LIN {X 0,Y 185.683,Z 170.354,A -85,B 0,C 180,E1 -22212.634,E2 -22212.634} C_VEL
LIN {X 0,Y 186.754,Z 173.291,A -85,B 0,C 180,E1 -22212.96,E2 -22212.96} C_VEL
LIN {X 0,Y 193.586,Z 186.24,A -85,B 0,C 180,E1 -22214.699,E2 -22214.699} C_VEL
LIN {X 0,Y 199.796,Z 199.622,A -85,B 0,C 180,E1 -22216.226,E2 -22216.226} C_VEL
LIN {X 0,Y 202.678,Z 207.739,A -85,B 0,C 180,E1 -22216.973,E2 -22216.973} C_VEL
LIN {X 0,Y 199.951,Z 270.572,A -85,B 0,C 180,E1 -22219.192,E2 -22219.192} C_VEL
LIN {X 0,Y 198.885,Z 284.057,A -85,B 0,C 180,E1 -22220.081,E2 -22220.081} C_VEL
LIN {X 0,Y 197.521,Z 296.496,A -85,B 0,C 180,E1 -22221.303,E2 -22221.303} C_VEL
LIN {X 0,Y 195.797,Z 307.712,A -85,B 0,C 180,E1 -22222.783,E2 -22222.783} C_VEL
LIN {X 0,Y 193.672,Z 319.403,A -85,B 0,C 180,E1 -22224.795,E2 -22224.795} C_VEL
LIN {X 0,Y 191.562,Z 329.915,A -85,B 0,C 180,E1 -22227.109,E2 -22227.109} C_VEL
LIN {X 0,Y 189.509,Z 339.066,A -85,B 0,C 180,E1 -22229.646,E2 -22229.646} C_VEL
LIN {X 0,Y 187.491,Z 347.803,A -85,B 0,C 180,E1 -22232.686,E2 -22232.686} C_VEL
LIN {X 0,Y 185.853,Z 355.279,A -85,B 0,C 180,E1 -22235.969,E2 -22235.969} C_VEL
LIN {X 0,Y 184.768,Z 360.328,A -85,B 0,C 180,E1 -22238.752,E2 -22238.752} C_VEL
LIN {X 0,Y 183.841,Z 365.228,A -85,B 0,C 180,E1 -22242.138,E2 -22242.138} C_VEL
LIN {X 0,Y 183.252,Z 368.971,A -85,B 0,C 180,E1 -22245.573,E2 -22245.573} C_VEL
LIN {X 0,Y 183.005,Z 370.856,A -85,B 0,C 180,E1 -22247.893,E2 -22247.893} C_VEL
LIN {X 0,Y 182.982,Z 372.28,A -85,B 0,C 180,E1 -22250.223,E2 -22250.223} C_VEL
LIN {X 0,Y 183.211,Z 373.408,A -85,B 0,C 180,E1 -22252.981,E2 -22252.981} C_VEL
LIN {X 0,Y 184.045,Z 373.895,A -85,B 0,C 180,E1 -22257.274,E2 -22257.274} C_VEL
LIN {X 0,Y 184.848,Z 373.552,A -85,B 0,C 180,E1 -22259.622,E2 -22259.622} C_VEL
LIN {X 0,Y 185.845,Z 372.724,A -85,B 0,C 180,E1 -22261.967,E2 -22261.967} C_VEL
LIN {X 0,Y 187.135,Z 371.423,A -85,B 0,C 180,E1 -22264.287,E2 -22264.287} C_VEL
LIN {X 0,Y 189.469,Z 368.561,A -85,B 0,C 180,E1 -22267.737,E2 -22267.737} C_VEL
LIN {X 0,Y 192.379,Z 364.501,A -85,B 0,C 180,E1 -22271.116,E2 -22271.116} C_VEL
LIN {X 0,Y 196.276,Z 358.58,A -85,B 0,C 180,E1 -22274.64,E2 -22274.64} C_VEL
LIN {X 0,Y 200.108,Z 352.117,A -85,B 0,C 180,E1 -22277.523,E2 -22277.523} C_VEL
LIN {X 0,Y 204.75,Z 343.271,A -85,B 0,C 180,E1 -22280.562,E2 -22280.562} C_VEL
LIN {X 0,Y 209,Z 334.332,A -85,B 0,C 180,E1 -22282.876,E2 -22282.876} C_VEL
LIN {X 0,Y 213.308,Z 323.651,A -85,B 0,C 180,E1 -22285.043,E2 -22285.043} C_VEL
LIN {X 0,Y 216.807,Z 313.421,A -85,B 0,C 180,E1 -22286.659,E2 -22286.659} C_VEL
LIN {X 0,Y 219.931,Z 301.93,A -85,B 0,C 180,E1 -22288.084,E2 -22288.084} C_VEL
LIN {X 0,Y 222.4,Z 290.554,A -85,B 0,C 180,E1 -22289.133,E2 -22289.133} C_VEL
LIN {X 0,Y 224.406,Z 278.014,A -85,B 0,C 180,E1 -22289.955,E2 -22289.955} C_VEL
LIN {X 0,Y 225.625,Z 265.738,A -85,B 0,C 180,E1 -22290.474,E2 -22290.474} C_VEL
LIN {X 0,Y 227.824,Z 230.741,A -85,B 0,C 180,E1 -22291.554,E2 -22291.554} C_VEL
LIN {X 0,Y 224.167,Z 223.088,A -85,B 0,C 180,E1 -22293.044,E2 -22293.044} C_VEL
LIN {X 0,Y 217.84,Z 212.554,A -85,B 0,C 180,E1 -22295.719,E2 -22295.719} C_VEL
LIN {X 0,Y 212.058,Z 203.914,A -85,B 0,C 180,E1 -22298.467,E2 -22298.467} C_VEL
LIN {X 0,Y 206.963,Z 196.712,A -85,B 0,C 180,E1 -22301.18,E2 -22301.18} C_VEL
LIN {X 0,Y 204.092,Z 192.954,A -85,B 0,C 180,E1 -22302.853,E2 -22302.853} C_VEL
LIN {X 0,Y 200.713,Z 188.672,A -85,B 0,C 180,E1 -22305.051,E2 -22305.051} C_VEL
LIN {X 0,Y 199.927,Z 187.365,A -85,B 0,C 180,E1 -22305.625,E2 -22305.625} C_VEL
LIN {X 0,Y 197.269,Z 184.822,A -85,B 0,C 180,E1 -22307.527,E2 -22307.527} C_VEL
LIN {X 0,Y 195.63,Z 181.953,A -85,B 0,C 180,E1 -22308.932,E2 -22308.932} C_VEL
LIN {X 0,Y 192.955,Z 179.723,A -85,B 0,C 180,E1 -22311.217,E2 -22311.217} C_VEL
LIN {X 0,Y 191.565,Z 177.134,A -85,B 0,C 180,E1 -22312.756,E2 -22312.756} C_VEL
LIN {X 0,Y 191.264,Z 176.32,A -85,B 0,C 180,E1 -22313.143,E2 -22313.143} C_VEL
LIN {X 0,Y 188.409,Z 174.865,A -85,B 0,C 180,E1 -22316.391,E2 -22316.391} C_VEL
LIN {X 0,Y 186.674,Z 171.895,A -85,B 0,C 180,E1 -22319.259,E2 -22319.259} C_VEL
LIN {X 0,Y 186.346,Z 170.267,A -85,B 0,C 180,E1 -22320.135,E2 -22320.135} C_VEL
LIN {X 0,Y 185.885,Z 170.317,A -85,B 0,C 180,E1 -22324.337,E2 -22324.337} C_VEL
LIN {X 0,Y 185.976,Z 170.302,A -85,B 0,C 180,E1 -22328.695,E2 -22328.695} C_VEL
LIN {X 0,Y 185.723,Z 170.332,A -85,B 0,C 180,E1 -22333.124,E2 -22333.124} C_VEL
LIN {X 0,Y 185.682,Z 170.347,A -85,B 0,C 180,E1 -22336.492,E2 -22336.492} C_VEL
LIN {X 0,Y 185.915,Z 171.497,A -85,B 0,C 180,E1 -22338.814,E2 -22338.814} C_VEL
LIN {X 0,Y 186.795,Z 173.557,A -85,B 0,C 180,E1 -22340.655,E2 -22340.655} C_VEL
LIN {X 0,Y 188.885,Z 175.776,A -85,B 0,C 180,E1 -22343.723,E2 -22343.723} C_VEL
LIN {X 0,Y 191.922,Z 179.165,A -85,B 0,C 180,E1 -22347.242,E2 -22347.242} C_VEL
LIN {X 0,Y 194.898,Z 183.776,A -85,B 0,C 180,E1 -22350.131,E2 -22350.131} C_VEL
LIN {X 0,Y 197.691,Z 187.166,A -85,B 0,C 180,E1 -22352.379,E2 -22352.379} C_VEL
LIN {X 0,Y 202.172,Z 193.838,A -85,B 0,C 180,E1 -22355.611,E2 -22355.611} C_VEL
LIN {X 0,Y 206.17,Z 199.973,A -85,B 0,C 180,E1 -22358.086,E2 -22358.086} C_VEL
LIN {X 0,Y 209.889,Z 206.05,A -85,B 0,C 180,E1 -22360.173,E2 -22360.173} C_VEL
LIN {X 0,Y 213.804,Z 212.78,A -85,B 0,C 180,E1 -22362.196,E2 -22362.196} C_VEL
LIN {X 0,Y 219.154,Z 223.042,A -85,B 0,C 180,E1 -22364.732,E2 -22364.732} C_VEL
LIN {X 0,Y 224.276,Z 234.48,A -85,B 0,C 180,E1 -22366.986,E2 -22366.986} C_VEL
LIN {X 0,Y 226.38,Z 239.916,A -85,B 0,C 180,E1 -22367.89,E2 -22367.89} C_VEL
LIN {X 0,Y 226.931,Z 246.644,A -85,B 0,C 180,E1 -22368.381,E2 -22368.381} C_VEL
LIN {X 0,Y 225.009,Z 277.037,A -85,B 0,C 180,E1 -22369.312,E2 -22369.312} C_VEL
LIN {X 0,Y 224.097,Z 282.869,A -85,B 0,C 180,E1 -22369.364,E2 -22369.364} C_VEL
LIN {X 0,Y 221.088,Z 292.299,A -85,B 0,C 180,E1 -22369.24,E2 -22369.24} C_VEL
LIN {X 0,Y 217.548,Z 301.55,A -85,B 0,C 180,E1 -22369.224,E2 -22369.224} C_VEL
LIN {X 0,Y 215.797,Z 307.1,A -85,B 0,C 180,E1 -22369.487,E2 -22369.487} C_VEL
LIN {X 0,Y 212.279,Z 320.078,A -85,B 0,C 180,E1 -22370.715,E2 -22370.715} C_VEL
LIN {X 0,Y 208.678,Z 330.767,A -85,B 0,C 180,E1 -22372.074,E2 -22372.074} C_VEL
LIN {X 0,Y 204.289,Z 341.732,A -85,B 0,C 180,E1 -22373.904,E2 -22373.904} C_VEL
LIN {X 0,Y 199.37,Z 352.427,A -85,B 0,C 180,E1 -22376.275,E2 -22376.275} C_VEL
LIN {X 0,Y 195.224,Z 360.362,A -85,B 0,C 180,E1 -22378.533,E2 -22378.533} C_VEL
LIN {X 0,Y 190.711,Z 368.187,A -85,B 0,C 180,E1 -22381.375,E2 -22381.375} C_VEL
LIN {X 0,Y 186.739,Z 374.659,A -85,B 0,C 180,E1 -22384.473,E2 -22384.473} C_VEL
LIN {X 0,Y 183.642,Z 379.535,A -85,B 0,C 180,E1 -22387.498,E2 -22387.498} C_VEL
LIN {X 0,Y 180.899,Z 383.498,A -85,B 0,C 180,E1 -22390.717,E2 -22390.717} C_VEL
LIN {X 0,Y 178.676,Z 386.462,A -85,B 0,C 180,E1 -22394.017,E2 -22394.017} C_VEL
LIN {X 0,Y 176.939,Z 388.948,A -85,B 0,C 180,E1 -22398.545,E2 -22398.545} C_VEL
LIN {X 0,Y 176.128,Z 389.914,A -85,B 0,C 180,E1 -22403.124,E2 -22403.124} C_VEL
LIN {X 0,Y 176.125,Z 389.685,A -85,B 0,C 180,E1 -22406.027,E2 -22406.027} C_VEL
LIN {X 0,Y 176.394,Z 388.365,A -85,B 0,C 180,E1 -22410,E2 -22410} C_VEL
LIN {X 0,Y 176.229,Z 387.022,A -85,B 0,C 180,E1 -22412.285,E2 -22412.285} C_VEL
LIN {X 0,Y 176.169,Z 384.135,A -85,B 0,C 180,E1 -22415.723,E2 -22415.723} C_VEL
LIN {X 0,Y 176.448,Z 380.179,A -85,B 0,C 180,E1 -22419.167,E2 -22419.167} C_VEL
LIN {X 0,Y 177.299,Z 374.04,A -85,B 0,C 180,E1 -22423.175,E2 -22423.175} C_VEL
LIN {X 0,Y 178.698,Z 367.3,A -85,B 0,C 180,E1 -22426.566,E2 -22426.566} C_VEL
LIN {X 0,Y 180.547,Z 358.895,A -85,B 0,C 180,E1 -22429.913,E2 -22429.913} C_VEL
LIN {X 0,Y 181.898,Z 352.509,A -85,B 0,C 180,E1 -22431.983,E2 -22431.983} C_VEL
LIN {X 0,Y 183.957,Z 344.092,A -85,B 0,C 180,E1 -22434.248,E2 -22434.248} C_VEL
LIN {X 0,Y 186.267,Z 333.179,A -85,B 0,C 180,E1 -22436.618,E2 -22436.618} C_VEL
LIN {X 0,Y 188.393,Z 322.564,A -85,B 0,C 180,E1 -22438.401,E2 -22438.401} C_VEL
LIN {X 0,Y 190.53,Z 309.778,A -85,B 0,C 180,E1 -22440.018,E2 -22440.018} C_VEL
LIN {X 0,Y 192.193,Z 297.008,A -85,B 0,C 180,E1 -22441.175,E2 -22441.175} C_VEL
LIN {X 0,Y 193.255,Z 284.752,A -85,B 0,C 180,E1 -22441.9,E2 -22441.9} C_VEL
LIN {X 0,Y 195.225,Z 238.101,A -85,B 0,C 180,E1 -22443.6,E2 -22443.6} C_VEL
LIN {X 0,Y 192.063,Z 207.786,A -85,B 0,C 180,E1 -22445.365,E2 -22445.365} C_VEL
LIN {X 0,Y 185.656,Z 190.417,A -85,B 0,C 180,E1 -22447.212,E2 -22447.212} C_VEL
LIN {X 0,Y 180.83,Z 179.385,A -85,B 0,C 180,E1 -22448.597,E2 -22448.597} C_VEL
LIN {X 0,Y 179.797,Z 176.7,A -85,B 0,C 180,E1 -22449.002,E2 -22449.002} C_VEL
LIN {X 0,Y 178.427,Z 171.261,A -85,B 0,C 180,E1 -22452.036,E2 -22452.036} C_VEL
LIN {X 0,Y 178.395,Z 171.266,A -85,B 0,C 180,E1 -22455.163,E2 -22455.163} C_VEL
LIN {X 0,Y 178.404,Z 171.265,A -85,B 0,C 180,E1 -22458.458,E2 -22458.458} C_VEL
LIN {X 0,Y 178.423,Z 171.263,A -85,B 0,C 180,E1 -22463.783,E2 -22463.783} C_VEL
LIN {X 0,Y 178.488,Z 171.252,A -85,B 0,C 180,E1 -22466.546,E2 -22466.546} C_VEL
LIN {X 0,Y 178.524,Z 171.248,A -85,B 0,C 180,E1 -22470.006,E2 -22470.006} C_VEL
LIN {X 0,Y 178.52,Z 171.248,A -85,B 0,C 180,E1 -22474.885,E2 -22474.885} C_VEL
LIN {X 0,Y 178.589,Z 171.197,A -85,B 0,C 180,E1 -22480.815,E2 -22480.815} C_VEL
LIN {X 0,Y 178.643,Z 171.22,A -85,B 0,C 180,E1 -22486.346,E2 -22486.346} C_VEL
LIN {X 0,Y 178.905,Z 171.195,A -85,B 0,C 180,E1 -22490.959,E2 -22490.959} C_VEL
LIN {X 0,Y 179.149,Z 171.165,A -85,B 0,C 180,E1 -22497.751,E2 -22497.751} C_VEL
LIN {X 0,Y 179.37,Z 171.135,A -85,B 0,C 180,E1 -22500,E2 -22500} C_VEL
LIN {X 0,Y 178.867,Z 171.194,A -85,B 0,C 180,E1 -22504.507,E2 -22504.507} C_VEL
LIN {X 0,Y 178.911,Z 171.191,A -85,B 0,C 180,E1 -22509.04,E2 -22509.04} C_VEL
LIN {X 0,Y 178.657,Z 171.222,A -85,B 0,C 180,E1 -22513.652,E2 -22513.652} C_VEL
LIN {X 0,Y 178.622,Z 171.227,A -85,B 0,C 180,E1 -22519.215,E2 -22519.215} C_VEL
LIN {X 0,Y 178.519,Z 171.246,A -85,B 0,C 180,E1 -22525.114,E2 -22525.114} C_VEL
LIN {X 0,Y 178.52,Z 171.232,A -85,B 0,C 180,E1 -22529.993,E2 -22529.993} C_VEL
LIN {X 0,Y 178.483,Z 171.25,A -85,B 0,C 180,E1 -22534.219,E2 -22534.219} C_VEL
LIN {X 0,Y 178.394,Z 171.25,A -85,B 0,C 180,E1 -22539.074,E2 -22539.074} C_VEL
LIN {X 0,Y 178.397,Z 171.261,A -85,B 0,C 180,E1 -22542.045,E2 -22542.045} C_VEL
LIN {X 0,Y 178.393,Z 171.253,A -85,B 0,C 180,E1 -22545.164,E2 -22545.164} C_VEL
LIN {X 0,Y 178.402,Z 171.261,A -85,B 0,C 180,E1 -22548.459,E2 -22548.459} C_VEL
LIN {X 0,Y 178.422,Z 171.261,A -85,B 0,C 180,E1 -22553.783,E2 -22553.783} C_VEL
LIN {X 0,Y 178.486,Z 171.242,A -85,B 0,C 180,E1 -22556.547,E2 -22556.547} C_VEL
LIN {X 0,Y 178.522,Z 171.233,A -85,B 0,C 180,E1 -22560.006,E2 -22560.006} C_VEL
LIN {X 0,Y 178.519,Z 171.237,A -85,B 0,C 180,E1 -22564.886,E2 -22564.886} C_VEL
LIN {X 0,Y 178.624,Z 171.226,A -85,B 0,C 180,E1 -22571.288,E2 -22571.288} C_VEL
LIN {X 0,Y 179.695,Z 174.19,A -85,B 0,C 180,E1 -22571.687,E2 -22571.687} C_VEL
LIN {X 0,Y 184.03,Z 181.923,A -85,B 0,C 180,E1 -22572.86,E2 -22572.86} C_VEL
LIN {X 0,Y 192.925,Z 200.17,A -85,B 0,C 180,E1 -22575.192,E2 -22575.192} C_VEL
LIN {X 0,Y 196.304,Z 209.181,A -85,B 0,C 180,E1 -22576.1,E2 -22576.1} C_VEL
LIN {X 0,Y 193.535,Z 270.405,A -85,B 0,C 180,E1 -22578.313,E2 -22578.313} C_VEL
LIN {X 0,Y 192.39,Z 284.408,A -85,B 0,C 180,E1 -22579.257,E2 -22579.257} C_VEL
LIN {X 0,Y 190.855,Z 297.508,A -85,B 0,C 180,E1 -22580.596,E2 -22580.596} C_VEL
LIN {X 0,Y 188.946,Z 309.37,A -85,B 0,C 180,E1 -22582.251,E2 -22582.251} C_VEL
LIN {X 0,Y 186.759,Z 320.819,A -85,B 0,C 180,E1 -22584.331,E2 -22584.331} C_VEL
LIN {X 0,Y 184.559,Z 331.091,A -85,B 0,C 180,E1 -22586.726,E2 -22586.726} C_VEL
LIN {X 0,Y 182.317,Z 340.478,A -85,B 0,C 180,E1 -22589.481,E2 -22589.481} C_VEL
LIN {X 0,Y 180.259,Z 349.401,A -85,B 0,C 180,E1 -22592.794,E2 -22592.794} C_VEL
LIN {X 0,Y 178.58,Z 356.596,A -85,B 0,C 180,E1 -22596.213,E2 -22596.213} C_VEL
LIN {X 0,Y 177.519,Z 361.503,A -85,B 0,C 180,E1 -22599.112,E2 -22599.112} C_VEL
LIN {X 0,Y 176.617,Z 366.201,A -85,B 0,C 180,E1 -22602.642,E2 -22602.642} C_VEL
LIN {X 0,Y 176.025,Z 370.083,A -85,B 0,C 180,E1 -22606.62,E2 -22606.62} C_VEL
LIN {X 0,Y 175.943,Z 372.894,A -85,B 0,C 180,E1 -22611.07,E2 -22611.07} C_VEL
LIN {X 0,Y 176.181,Z 373.768,A -85,B 0,C 180,E1 -22613.51,E2 -22613.51} C_VEL
LIN {X 0,Y 176.593,Z 374.196,A -85,B 0,C 180,E1 -22615.963,E2 -22615.963} C_VEL
LIN {X 0,Y 177.676,Z 374.027,A -85,B 0,C 180,E1 -22619.518,E2 -22619.518} C_VEL
LIN {X 0,Y 179.353,Z 372.789,A -85,B 0,C 180,E1 -22623.271,E2 -22623.271} C_VEL
LIN {X 0,Y 180.795,Z 371.406,A -85,B 0,C 180,E1 -22625.669,E2 -22625.669} C_VEL
LIN {X 0,Y 183.351,Z 368.412,A -85,B 0,C 180,E1 -22629.18,E2 -22629.18} C_VEL
LIN {X 0,Y 186.612,Z 364.099,A -85,B 0,C 180,E1 -22632.68,E2 -22632.68} C_VEL
LIN {X 0,Y 190.53,Z 358.405,A -85,B 0,C 180,E1 -22636.038,E2 -22636.038} C_VEL
LIN {X 0,Y 194.945,Z 351.263,A -85,B 0,C 180,E1 -22639.208,E2 -22639.208} C_VEL
LIN {X 0,Y 199.065,Z 343.785,A -85,B 0,C 180,E1 -22641.771,E2 -22641.771} C_VEL
LIN {X 0,Y 203.726,Z 334.428,A -85,B 0,C 180,E1 -22644.224,E2 -22644.224} C_VEL
LIN {X 0,Y 207.99,Z 324.269,A -85,B 0,C 180,E1 -22646.314,E2 -22646.314} C_VEL
LIN {X 0,Y 211.87,Z 313.396,A -85,B 0,C 180,E1 -22648.047,E2 -22648.047} C_VEL
LIN {X 0,Y 215.169,Z 301.7,A -85,B 0,C 180,E1 -22649.484,E2 -22649.484} C_VEL
LIN {X 0,Y 217.846,Z 289.592,A -85,B 0,C 180,E1 -22650.582,E2 -22650.582} C_VEL
LIN {X 0,Y 219.859,Z 276.83,A -85,B 0,C 180,E1 -22651.4,E2 -22651.4} C_VEL
LIN {X 0,Y 221.194,Z 262.498,A -85,B 0,C 180,E1 -22651.941,E2 -22651.941} C_VEL
LIN {X 0,Y 223.096,Z 233.455,A -85,B 0,C 180,E1 -22652.844,E2 -22652.844} C_VEL
LIN {X 0,Y 219.833,Z 226.818,A -85,B 0,C 180,E1 -22654.245,E2 -22654.245} C_VEL
LIN {X 0,Y 214.285,Z 217.443,A -85,B 0,C 180,E1 -22656.756,E2 -22656.756} C_VEL
LIN {X 0,Y 208.779,Z 209.045,A -85,B 0,C 180,E1 -22659.527,E2 -22659.527} C_VEL
LIN {X 0,Y 204.268,Z 202.61,A -85,B 0,C 180,E1 -22662.058,E2 -22662.058} C_VEL
LIN {X 0,Y 200.956,Z 198.121,A -85,B 0,C 180,E1 -22664.144,E2 -22664.144} C_VEL
LIN {X 0,Y 198.215,Z 194.314,A -85,B 0,C 180,E1 -22666.072,E2 -22666.072} C_VEL
LIN {X 0,Y 194.988,Z 190.63,A -85,B 0,C 180,E1 -22668.538,E2 -22668.538} C_VEL
LIN {X 0,Y 193.865,Z 188.579,A -85,B 0,C 180,E1 -22669.557,E2 -22669.557} C_VEL
LIN {X 0,Y 191.372,Z 186.351,A -85,B 0,C 180,E1 -22671.811,E2 -22671.811} C_VEL
LIN {X 0,Y 189.821,Z 183.428,A -85,B 0,C 180,E1 -22673.623,E2 -22673.623} C_VEL
LIN {X 0,Y 186.829,Z 181.328,A -85,B 0,C 180,E1 -22677.305,E2 -22677.305} C_VEL
LIN {X 0,Y 185.305,Z 178.253,A -85,B 0,C 180,E1 -22680.136,E2 -22680.136} C_VEL
LIN {X 0,Y 185.063,Z 177.272,A -85,B 0,C 180,E1 -22680.816,E2 -22680.816} C_VEL
LIN {X 0,Y 182.802,Z 176.663,A -85,B 0,C 180,E1 -22688.847,E2 -22688.847} C_VEL
LIN {X 0,Y 184.131,Z 177.385,A -85,B 0,C 180,E1 -22696.635,E2 -22696.635} C_VEL
LIN {X 0,Y 184.769,Z 178.417,A -85,B 0,C 180,E1 -22698.331,E2 -22698.331} C_VEL
LIN {X 0,Y 185.917,Z 180.829,A -85,B 0,C 180,E1 -22700.757,E2 -22700.757} C_VEL
LIN {X 0,Y 187.603,Z 182.649,A -85,B 0,C 180,E1 -22703.284,E2 -22703.284} C_VEL
LIN {X 0,Y 190.562,Z 186.17,A -85,B 0,C 180,E1 -22706.859,E2 -22706.859} C_VEL
LIN {X 0,Y 193.141,Z 190.298,A -85,B 0,C 180,E1 -22709.484,E2 -22709.484} C_VEL
LIN {X 0,Y 195.738,Z 193.586,A -85,B 0,C 180,E1 -22711.677,E2 -22711.677} C_VEL
LIN {X 0,Y 199.913,Z 200.03,A -85,B 0,C 180,E1 -22714.84,E2 -22714.84} C_VEL
LIN {X 0,Y 203.71,Z 206.099,A -85,B 0,C 180,E1 -22717.331,E2 -22717.331} C_VEL
LIN {X 0,Y 206.999,Z 211.66,A -85,B 0,C 180,E1 -22719.273,E2 -22719.273} C_VEL
LIN {X 0,Y 211.426,Z 219.589,A -85,B 0,C 180,E1 -22721.669,E2 -22721.669} C_VEL
LIN {X 0,Y 216.84,Z 230.662,A -85,B 0,C 180,E1 -22724.358,E2 -22724.358} C_VEL
LIN {X 0,Y 221.216,Z 241.243,A -85,B 0,C 180,E1 -22726.381,E2 -22726.381} C_VEL
LIN {X 0,Y 221.895,Z 242.935,A -85,B 0,C 180,E1 -22726.683,E2 -22726.683} C_VEL
LIN {X 0,Y 222.294,Z 247.076,A -85,B 0,C 180,E1 -22727.02,E2 -22727.02} C_VEL
LIN {X 0,Y 219.532,Z 285.815,A -85,B 0,C 180,E1 -22728.25,E2 -22728.25} C_VEL
LIN {X 0,Y 217.473,Z 299.233,A -85,B 0,C 180,E1 -22728.932,E2 -22728.932} C_VEL
LIN {X 0,Y 215.797,Z 307.1,A -85,B 0,C 180,E1 -22729.487,E2 -22729.487} C_VEL
LIN {X 0,Y 213.849,Z 312.694,A -85,B 0,C 180,E1 -22729.811,E2 -22729.811} C_VEL
LIN {X 0,Y 209.199,Z 321.494,A -85,B 0,C 180,E1 -22730.134,E2 -22730.134} C_VEL
LIN {X 0,Y 204.327,Z 329.786,A -85,B 0,C 180,E1 -22730.653,E2 -22730.653} C_VEL
LIN {X 0,Y 202.043,Z 334.607,A -85,B 0,C 180,E1 -22731.281,E2 -22731.281} C_VEL
LIN {X 0,Y 197.677,Z 344.642,A -85,B 0,C 180,E1 -22733.133,E2 -22733.133} C_VEL
LIN {X 0,Y 192.711,Z 354.666,A -85,B 0,C 180,E1 -22735.578,E2 -22735.578} C_VEL
LIN {X 0,Y 187.604,Z 363.522,A -85,B 0,C 180,E1 -22738.367,E2 -22738.367} C_VEL
LIN {X 0,Y 183.06,Z 370.68,A -85,B 0,C 180,E1 -22741.321,E2 -22741.321} C_VEL
LIN {X 0,Y 179.28,Z 376.429,A -85,B 0,C 180,E1 -22744.455,E2 -22744.455} C_VEL
LIN {X 0,Y 176.033,Z 381.002,A -85,B 0,C 180,E1 -22747.71,E2 -22747.71} C_VEL
LIN {X 0,Y 173.346,Z 384.521,A -85,B 0,C 180,E1 -22751.074,E2 -22751.074} C_VEL
LIN {X 0,Y 171.842,Z 386.314,A -85,B 0,C 180,E1 -22753.364,E2 -22753.364} C_VEL
LIN {X 0,Y 169.967,Z 388.718,A -85,B 0,C 180,E1 -22758.068,E2 -22758.068} C_VEL
LIN {X 0,Y 169.371,Z 389.351,A -85,B 0,C 180,E1 -22760.445,E2 -22760.445} C_VEL
LIN {X 0,Y 169.079,Z 389.581,A -85,B 0,C 180,E1 -22762.836,E2 -22762.836} C_VEL
LIN {X 0,Y 169.144,Z 388.853,A -85,B 0,C 180,E1 -22767.618,E2 -22767.618} C_VEL
LIN {X 0,Y 169.309,Z 387.903,A -85,B 0,C 180,E1 -22770,E2 -22770} C_VEL
LIN {X 0,Y 169.1,Z 385.236,A -85,B 0,C 180,E1 -22774.07,E2 -22774.07} C_VEL
LIN {X 0,Y 169.266,Z 380.947,A -85,B 0,C 180,E1 -22778.355,E2 -22778.355} C_VEL
LIN {X 0,Y 169.863,Z 376.113,A -85,B 0,C 180,E1 -22781.939,E2 -22781.939} C_VEL
LIN {X 0,Y 171.019,Z 369.981,A -85,B 0,C 180,E1 -22785.492,E2 -22785.492} C_VEL
LIN {X 0,Y 172.699,Z 362.32,A -85,B 0,C 180,E1 -22788.999,E2 -22788.999} C_VEL
LIN {X 0,Y 174.757,Z 353.387,A -85,B 0,C 180,E1 -22792.212,E2 -22792.212} C_VEL
LIN {X 0,Y 177.197,Z 343.797,A -85,B 0,C 180,E1 -22794.923,E2 -22794.923} C_VEL
LIN {X 0,Y 179.589,Z 332.885,A -85,B 0,C 180,E1 -22797.375,E2 -22797.375} C_VEL
LIN {X 0,Y 181.81,Z 322.285,A -85,B 0,C 180,E1 -22799.211,E2 -22799.211} C_VEL
LIN {X 0,Y 184.024,Z 309.51,A -85,B 0,C 180,E1 -22800.876,E2 -22800.876} C_VEL
LIN {X 0,Y 185.736,Z 296.808,A -85,B 0,C 180,E1 -22802.062,E2 -22802.062} C_VEL
LIN {X 0,Y 186.848,Z 284.399,A -85,B 0,C 180,E1 -22802.819,E2 -22802.819} C_VEL
LIN {X 0,Y 188.863,Z 238.895,A -85,B 0,C 180,E1 -22804.524,E2 -22804.524} C_VEL
LIN {X 0,Y 186.023,Z 210.18,A -85,B 0,C 180,E1 -22806.256,E2 -22806.256} C_VEL
LIN {X 0,Y 180.087,Z 193.89,A -85,B 0,C 180,E1 -22808.058,E2 -22808.058} C_VEL
LIN {X 0,Y 174.201,Z 180.352,A -85,B 0,C 180,E1 -22809.86,E2 -22809.86} C_VEL
LIN {X 0,Y 172.459,Z 176.4,A -85,B 0,C 180,E1 -22810.468,E2 -22810.468} C_VEL
LIN {X 0,Y 171.332,Z 172.144,A -85,B 0,C 180,E1 -22813.009,E2 -22813.009} C_VEL
LIN {X 0,Y 171.337,Z 172.146,A -85,B 0,C 180,E1 -22817.589,E2 -22817.589} C_VEL
LIN {X 0,Y 171.388,Z 172.139,A -85,B 0,C 180,E1 -22822.04,E2 -22822.04} C_VEL
LIN {X 0,Y 171.399,Z 172.136,A -85,B 0,C 180,E1 -22825.092,E2 -22825.092} C_VEL
LIN {X 0,Y 171.45,Z 172.129,A -85,B 0,C 180,E1 -22830.534,E2 -22830.534} C_VEL
LIN {X 0,Y 171.444,Z 172.128,A -85,B 0,C 180,E1 -22835.799,E2 -22835.799} C_VEL
LIN {X 0,Y 171.545,Z 172.072,A -85,B 0,C 180,E1 -22840.867,E2 -22840.867} C_VEL
LIN {X 0,Y 171.558,Z 172.097,A -85,B 0,C 180,E1 -22845.771,E2 -22845.771} C_VEL
LIN {X 0,Y 171.843,Z 172.077,A -85,B 0,C 180,E1 -22850.584,E2 -22850.584} C_VEL
LIN {X 0,Y 171.807,Z 172.073,A -85,B 0,C 180,E1 -22855.307,E2 -22855.307} C_VEL
LIN {X 0,Y 172.332,Z 172.011,A -85,B 0,C 180,E1 -22860,E2 -22860} C_VEL
LIN {X 0,Y 171.815,Z 172.074,A -85,B 0,C 180,E1 -22864.692,E2 -22864.692} C_VEL
LIN {X 0,Y 171.848,Z 172.07,A -85,B 0,C 180,E1 -22869.415,E2 -22869.415} C_VEL
LIN {X 0,Y 171.575,Z 172.106,A -85,B 0,C 180,E1 -22874.227,E2 -22874.227} C_VEL
LIN {X 0,Y 171.541,Z 172.106,A -85,B 0,C 180,E1 -22879.559,E2 -22879.559} C_VEL
LIN {X 0,Y 171.457,Z 172.126,A -85,B 0,C 180,E1 -22885.609,E2 -22885.609} C_VEL
LIN {X 0,Y 171.439,Z 172.113,A -85,B 0,C 180,E1 -22890.585,E2 -22890.585} C_VEL
LIN {X 0,Y 171.391,Z 172.132,A -85,B 0,C 180,E1 -22895.035,E2 -22895.035} C_VEL
LIN {X 0,Y 171.356,Z 172.125,A -85,B 0,C 180,E1 -22898.807,E2 -22898.807} C_VEL
LIN {X 0,Y 171.32,Z 172.135,A -85,B 0,C 180,E1 -22904.217,E2 -22904.217} C_VEL
LIN {X 0,Y 171.334,Z 172.142,A -85,B 0,C 180,E1 -22908.982,E2 -22908.982} C_VEL
LIN {X 0,Y 171.386,Z 172.13,A -85,B 0,C 180,E1 -22912.041,E2 -22912.041} C_VEL
LIN {X 0,Y 171.397,Z 172.134,A -85,B 0,C 180,E1 -22915.092,E2 -22915.092} C_VEL
LIN {X 0,Y 171.448,Z 172.119,A -85,B 0,C 180,E1 -22920.535,E2 -22920.535} C_VEL
LIN {X 0,Y 171.443,Z 172.115,A -85,B 0,C 180,E1 -22925.8,E2 -22925.8} C_VEL
LIN {X 0,Y 171.519,Z 172.118,A -85,B 0,C 180,E1 -22929.853,E2 -22929.853} C_VEL
LIN {X 0,Y 172.677,Z 175.19,A -85,B 0,C 180,E1 -22930.313,E2 -22930.313} C_VEL
LIN {X 0,Y 174.131,Z 177.575,A -85,B 0,C 180,E1 -22930.738,E2 -22930.738} C_VEL
LIN {X 0,Y 181.21,Z 190.789,A -85,B 0,C 180,E1 -22932.759,E2 -22932.759} C_VEL
LIN {X 0,Y 188.346,Z 206.211,A -85,B 0,C 180,E1 -22934.705,E2 -22934.705} C_VEL
LIN {X 0,Y 190.06,Z 211.072,A -85,B 0,C 180,E1 -22935.202,E2 -22935.202} C_VEL
LIN {X 0,Y 187.092,Z 271.113,A -85,B 0,C 180,E1 -22937.422,E2 -22937.422} C_VEL
LIN {X 0,Y 185.975,Z 284.449,A -85,B 0,C 180,E1 -22938.35,E2 -22938.35} C_VEL
LIN {X 0,Y 184.392,Z 297.494,A -85,B 0,C 180,E1 -22939.709,E2 -22939.709} C_VEL
LIN {X 0,Y 182.383,Z 309.432,A -85,B 0,C 180,E1 -22941.413,E2 -22941.413} C_VEL
LIN {X 0,Y 180.106,Z 320.927,A -85,B 0,C 180,E1 -22943.559,E2 -22943.559} C_VEL
LIN {X 0,Y 177.823,Z 331.246,A -85,B 0,C 180,E1 -22946.034,E2 -22946.034} C_VEL
LIN {X 0,Y 175.394,Z 341.035,A -85,B 0,C 180,E1 -22949.015,E2 -22949.015} C_VEL
LIN {X 0,Y 173.339,Z 349.607,A -85,B 0,C 180,E1 -22952.324,E2 -22952.324} C_VEL
LIN {X 0,Y 171.576,Z 356.834,A -85,B 0,C 180,E1 -22955.878,E2 -22955.878} C_VEL
LIN {X 0,Y 170.271,Z 362.604,A -85,B 0,C 180,E1 -22959.504,E2 -22959.504} C_VEL
LIN {X 0,Y 169.412,Z 367.131,A -85,B 0,C 180,E1 -22963.19,E2 -22963.19} C_VEL
LIN {X 0,Y 168.886,Z 370.541,A -85,B 0,C 180,E1 -22966.936,E2 -22966.936} C_VEL
LIN {X 0,Y 168.788,Z 372.24,A -85,B 0,C 180,E1 -22969.458,E2 -22969.458} C_VEL
LIN {X 0,Y 169.126,Z 374.091,A -85,B 0,C 180,E1 -22973.908,E2 -22973.908} C_VEL
LIN {X 0,Y 169.753,Z 374.581,A -85,B 0,C 180,E1 -22977.092,E2 -22977.092} C_VEL
LIN {X 0,Y 170.83,Z 374.352,A -85,B 0,C 180,E1 -22980.238,E2 -22980.238} C_VEL
LIN {X 0,Y 172.953,Z 372.859,A -85,B 0,C 180,E1 -22984.674,E2 -22984.674} C_VEL
LIN {X 0,Y 175.442,Z 370.412,A -85,B 0,C 180,E1 -22988.383,E2 -22988.383} C_VEL
LIN {X 0,Y 178.552,Z 366.806,A -85,B 0,C 180,E1 -22992.001,E2 -22992.001} C_VEL
LIN {X 0,Y 182.219,Z 362.075,A -85,B 0,C 180,E1 -22995.38,E2 -22995.38} C_VEL
LIN {X 0,Y 186.757,Z 355.541,A -85,B 0,C 180,E1 -22998.82,E2 -22998.82} C_VEL
LIN {X 0,Y 191.544,Z 347.772,A -85,B 0,C 180,E1 -23001.909,E2 -23001.909} C_VEL
LIN {X 0,Y 196.298,Z 339.029,A -85,B 0,C 180,E1 -23004.54,E2 -23004.54} C_VEL
LIN {X 0,Y 201.24,Z 328.565,A -85,B 0,C 180,E1 -23006.947,E2 -23006.947} C_VEL
LIN {X 0,Y 205.43,Z 318.125,A -85,B 0,C 180,E1 -23008.791,E2 -23008.791} C_VEL
LIN {X 0,Y 209.161,Z 306.296,A -85,B 0,C 180,E1 -23010.426,E2 -23010.426} C_VEL
LIN {X 0,Y 212.464,Z 293.334,A -85,B 0,C 180,E1 -23011.729,E2 -23011.729} C_VEL
LIN {X 0,Y 214.729,Z 280.833,A -85,B 0,C 180,E1 -23012.613,E2 -23012.613} C_VEL
LIN {X 0,Y 216.252,Z 267.769,A -85,B 0,C 180,E1 -23013.205,E2 -23013.205} C_VEL
LIN {X 0,Y 218.426,Z 236.071,A -85,B 0,C 180,E1 -23014.214,E2 -23014.214} C_VEL
LIN {X 0,Y 214.29,Z 228.217,A -85,B 0,C 180,E1 -23016.117,E2 -23016.117} C_VEL
LIN {X 0,Y 208.892,Z 219.259,A -85,B 0,C 180,E1 -23018.813,E2 -23018.813} C_VEL
LIN {X 0,Y 203.936,Z 211.728,A -85,B 0,C 180,E1 -23021.566,E2 -23021.566} C_VEL
LIN {X 0,Y 201.369,Z 208.122,A -85,B 0,C 180,E1 -23023.132,E2 -23023.132} C_VEL
LIN {X 0,Y 198.551,Z 204.136,A -85,B 0,C 180,E1 -23025.032,E2 -23025.032} C_VEL
LIN {X 0,Y 195.691,Z 200.125,A -85,B 0,C 180,E1 -23027.161,E2 -23027.161} C_VEL
LIN {X 0,Y 193.078,Z 197.016,A -85,B 0,C 180,E1 -23029.282,E2 -23029.282} C_VEL
LIN {X 0,Y 191.915,Z 195.099,A -85,B 0,C 180,E1 -23030.369,E2 -23030.369} C_VEL
LIN {X 0,Y 189.284,Z 192.184,A -85,B 0,C 180,E1 -23033.008,E2 -23033.008} C_VEL
LIN {X 0,Y 188.085,Z 189.991,A -85,B 0,C 180,E1 -23034.506,E2 -23034.506} C_VEL
LIN {X 0,Y 185.722,Z 188.301,A -85,B 0,C 180,E1 -23037.561,E2 -23037.561} C_VEL
LIN {X 0,Y 184.11,Z 185.046,A -85,B 0,C 180,E1 -23040.718,E2 -23040.718} C_VEL
LIN {X 0,Y 183.944,Z 184.296,A -85,B 0,C 180,E1 -23041.232,E2 -23041.232} C_VEL
LIN {X 0,Y 181.9,Z 183.708,A -85,B 0,C 180,E1 -23048.891,E2 -23048.891} C_VEL
LIN {X 0,Y 183.198,Z 184.46,A -85,B 0,C 180,E1 -23056.578,E2 -23056.578} C_VEL
LIN {X 0,Y 183.633,Z 185.328,A -85,B 0,C 180,E1 -23057.829,E2 -23057.829} C_VEL
LIN {X 0,Y 184.886,Z 187.861,A -85,B 0,C 180,E1 -23060.587,E2 -23060.587} C_VEL
LIN {X 0,Y 186.355,Z 189.526,A -85,B 0,C 180,E1 -23062.869,E2 -23062.869} C_VEL
LIN {X 0,Y 189.038,Z 192.936,A -85,B 0,C 180,E1 -23066.273,E2 -23066.273} C_VEL
LIN {X 0,Y 191.853,Z 197.329,A -85,B 0,C 180,E1 -23069.232,E2 -23069.232} C_VEL
LIN {X 0,Y 193.882,Z 200.175,A -85,B 0,C 180,E1 -23071.026,E2 -23071.026} C_VEL
LIN {X 0,Y 197.543,Z 205.961,A -85,B 0,C 180,E1 -23073.939,E2 -23073.939} C_VEL
LIN {X 0,Y 201.172,Z 212.047,A -85,B 0,C 180,E1 -23076.485,E2 -23076.485} C_VEL
LIN {X 0,Y 204.092,Z 217.144,A -85,B 0,C 180,E1 -23078.305,E2 -23078.305} C_VEL
LIN {X 0,Y 208.318,Z 225.011,A -85,B 0,C 180,E1 -23080.729,E2 -23080.729} C_VEL
LIN {X 0,Y 213.38,Z 235.709,A -85,B 0,C 180,E1 -23083.4,E2 -23083.4} C_VEL
LIN {X 0,Y 217.239,Z 245.41,A -85,B 0,C 180,E1 -23085.307,E2 -23085.307} C_VEL
LIN {X 0,Y 217.631,Z 247.159,A -85,B 0,C 180,E1 -23085.532,E2 -23085.532} C_VEL
LIN {X 0,Y 217.483,Z 251.734,A -85,B 0,C 180,E1 -23085.73,E2 -23085.73} C_VEL
LIN {X 0,Y 214.942,Z 285.552,A -85,B 0,C 180,E1 -23086.817,E2 -23086.817} C_VEL
LIN {X 0,Y 212.733,Z 299.39,A -85,B 0,C 180,E1 -23087.527,E2 -23087.527} C_VEL
LIN {X 0,Y 209.62,Z 312.431,A -85,B 0,C 180,E1 -23088.534,E2 -23088.534} C_VEL
LIN {X 0,Y 205.803,Z 324.693,A -85,B 0,C 180,E1 -23089.866,E2 -23089.866} C_VEL
LIN {X 0,Y 202.043,Z 334.607,A -85,B 0,C 180,E1 -23091.281,E2 -23091.281} C_VEL
LIN {X 0,Y 199.652,Z 339.399,A -85,B 0,C 180,E1 -23091.99,E2 -23091.99} C_VEL
LIN {X 0,Y 194.102,Z 346.912,A -85,B 0,C 180,E1 -23092.957,E2 -23092.957} C_VEL
LIN {X 0,Y 188.222,Z 353.89,A -85,B 0,C 180,E1 -23094.118,E2 -23094.118} C_VEL
LIN {X 0,Y 185.361,Z 357.845,A -85,B 0,C 180,E1 -23095.138,E2 -23095.138} C_VEL
LIN {X 0,Y 179.964,Z 366.38,A -85,B 0,C 180,E1 -23098.183,E2 -23098.183} C_VEL
LIN {X 0,Y 175.441,Z 372.916,A -85,B 0,C 180,E1 -23101.268,E2 -23101.268} C_VEL
LIN {X 0,Y 171.394,Z 378.594,A -85,B 0,C 180,E1 -23104.868,E2 -23104.868} C_VEL
LIN {X 0,Y 167.517,Z 383.39,A -85,B 0,C 180,E1 -23109.107,E2 -23109.107} C_VEL
LIN {X 0,Y 165.037,Z 386.178,A -85,B 0,C 180,E1 -23112.657,E2 -23112.657} C_VEL
LIN {X 0,Y 162.978,Z 388.493,A -85,B 0,C 180,E1 -23117.548,E2 -23117.548} C_VEL
LIN {X 0,Y 162.357,Z 389.07,A -85,B 0,C 180,E1 -23120.029,E2 -23120.029} C_VEL
LIN {X 0,Y 161.93,Z 389.023,A -85,B 0,C 180,E1 -23125.02,E2 -23125.02} C_VEL
LIN {X 0,Y 162.065,Z 388.431,A -85,B 0,C 180,E1 -23127.514,E2 -23127.514} C_VEL
LIN {X 0,Y 162.225,Z 387.44,A -85,B 0,C 180,E1 -23130,E2 -23130} C_VEL
LIN {X 0,Y 162.013,Z 384.975,A -85,B 0,C 180,E1 -23133.86,E2 -23133.86} C_VEL
LIN {X 0,Y 162.104,Z 381.665,A -85,B 0,C 180,E1 -23137.473,E2 -23137.473} C_VEL
LIN {X 0,Y 162.609,Z 377.142,A -85,B 0,C 180,E1 -23141.214,E2 -23141.214} C_VEL
LIN {X 0,Y 163.884,Z 370.238,A -85,B 0,C 180,E1 -23145.546,E2 -23145.546} C_VEL
LIN {X 0,Y 165.6,Z 362.703,A -85,B 0,C 180,E1 -23149.202,E2 -23149.202} C_VEL
LIN {X 0,Y 167.365,Z 354.979,A -85,B 0,C 180,E1 -23152.205,E2 -23152.205} C_VEL
LIN {X 0,Y 169.992,Z 345.676,A -85,B 0,C 180,E1 -23155.072,E2 -23155.072} C_VEL
LIN {X 0,Y 172.145,Z 336.537,A -85,B 0,C 180,E1 -23157.341,E2 -23157.341} C_VEL
LIN {X 0,Y 174.301,Z 326.846,A -85,B 0,C 180,E1 -23159.267,E2 -23159.267} C_VEL
LIN {X 0,Y 176.645,Z 314.579,A -85,B 0,C 180,E1 -23161.145,E2 -23161.145} C_VEL
LIN {X 0,Y 178.702,Z 301.792,A -85,B 0,C 180,E1 -23162.568,E2 -23162.568} C_VEL
LIN {X 0,Y 180.07,Z 289.247,A -85,B 0,C 180,E1 -23163.522,E2 -23163.522} C_VEL
LIN {X 0,Y 181.061,Z 272.951,A -85,B 0,C 180,E1 -23164.25,E2 -23164.25} C_VEL
LIN {X 0,Y 182.504,Z 238.965,A -85,B 0,C 180,E1 -23165.554,E2 -23165.554} C_VEL
LIN {X 0,Y 179.904,Z 212.035,A -85,B 0,C 180,E1 -23167.242,E2 -23167.242} C_VEL
LIN {X 0,Y 173.287,Z 194.162,A -85,B 0,C 180,E1 -23169.364,E2 -23169.364} C_VEL
LIN {X 0,Y 168.369,Z 183.186,A -85,B 0,C 180,E1 -23170.965,E2 -23170.965} C_VEL
LIN {X 0,Y 165.038,Z 175.993,A -85,B 0,C 180,E1 -23172.165,E2 -23172.165} C_VEL
LIN {X 0,Y 164.304,Z 173.02,A -85,B 0,C 180,E1 -23174.016,E2 -23174.016} C_VEL
LIN {X 0,Y 164.264,Z 173.026,A -85,B 0,C 180,E1 -23176.798,E2 -23176.798} C_VEL
LIN {X 0,Y 164.296,Z 173.023,A -85,B 0,C 180,E1 -23180.351,E2 -23180.351} C_VEL
LIN {X 0,Y 164.33,Z 173.016,A -85,B 0,C 180,E1 -23186.221,E2 -23186.221} C_VEL
LIN {X 0,Y 164.406,Z 173.006,A -85,B 0,C 180,E1 -23189.137,E2 -23189.137} C_VEL
LIN {X 0,Y 164.407,Z 173.005,A -85,B 0,C 180,E1 -23194.692,E2 -23194.692} C_VEL
LIN {X 0,Y 164.438,Z 172.963,A -85,B 0,C 180,E1 -23200.095,E2 -23200.095} C_VEL
LIN {X 0,Y 164.486,Z 172.971,A -85,B 0,C 180,E1 -23205.145,E2 -23205.145} C_VEL
LIN {X 0,Y 164.764,Z 172.958,A -85,B 0,C 180,E1 -23210.176,E2 -23210.176} C_VEL
LIN {X 0,Y 164.823,Z 172.939,A -85,B 0,C 180,E1 -23212.65,E2 -23212.65} C_VEL
LIN {X 0,Y 165.044,Z 172.922,A -85,B 0,C 180,E1 -23217.559,E2 -23217.559} C_VEL
LIN {X 0,Y 165.295,Z 172.887,A -85,B 0,C 180,E1 -23220,E2 -23220} C_VEL
LIN {X 0,Y 164.764,Z 172.953,A -85,B 0,C 180,E1 -23224.893,E2 -23224.893} C_VEL
LIN {X 0,Y 164.831,Z 172.948,A -85,B 0,C 180,E1 -23227.349,E2 -23227.349} C_VEL
LIN {X 0,Y 164.702,Z 172.949,A -85,B 0,C 180,E1 -23231.061,E2 -23231.061} C_VEL
LIN {X 0,Y 164.483,Z 172.994,A -85,B 0,C 180,E1 -23237.403,E2 -23237.403} C_VEL
LIN {X 0,Y 164.472,Z 172.982,A -85,B 0,C 180,E1 -23239.989,E2 -23239.989} C_VEL
LIN {X 0,Y 164.384,Z 173.008,A -85,B 0,C 180,E1 -23246.128,E2 -23246.128} C_VEL
LIN {X 0,Y 164.373,Z 172.995,A -85,B 0,C 180,E1 -23251.227,E2 -23251.227} C_VEL
LIN {X 0,Y 164.293,Z 173.011,A -85,B 0,C 180,E1 -23256.789,E2 -23256.789} C_VEL
LIN {X 0,Y 164.29,Z 173.009,A -85,B 0,C 180,E1 -23259.916,E2 -23259.916} C_VEL
LIN {X 0,Y 164.278,Z 173.017,A -85,B 0,C 180,E1 -23263.342,E2 -23263.342} C_VEL
LIN {X 0,Y 164.291,Z 173.014,A -85,B 0,C 180,E1 -23266.809,E2 -23266.809} C_VEL
LIN {X 0,Y 164.294,Z 173.015,A -85,B 0,C 180,E1 -23270.352,E2 -23270.352} C_VEL
LIN {X 0,Y 164.329,Z 173.015,A -85,B 0,C 180,E1 -23274.349,E2 -23274.349} C_VEL
LIN {X 0,Y 164.39,Z 172.986,A -85,B 0,C 180,E1 -23279.135,E2 -23279.135} C_VEL
LIN {X 0,Y 164.405,Z 172.995,A -85,B 0,C 180,E1 -23284.693,E2 -23284.693} C_VEL
LIN {X 0,Y 164.403,Z 173.008,A -85,B 0,C 180,E1 -23288.288,E2 -23288.288} C_VEL
LIN {X 0,Y 165.526,Z 175.982,A -85,B 0,C 180,E1 -23288.756,E2 -23288.756} C_VEL
LIN {X 0,Y 167.012,Z 178.314,A -85,B 0,C 180,E1 -23289.224,E2 -23289.224} C_VEL
LIN {X 0,Y 173.394,Z 189.782,A -85,B 0,C 180,E1 -23291.194,E2 -23291.194} C_VEL
LIN {X 0,Y 181.624,Z 206.927,A -85,B 0,C 180,E1 -23293.582,E2 -23293.582} C_VEL
LIN {X 0,Y 183.676,Z 212.172,A -85,B 0,C 180,E1 -23294.18,E2 -23294.18} C_VEL
LIN {X 0,Y 180.744,Z 271.142,A -85,B 0,C 180,E1 -23296.431,E2 -23296.431} C_VEL
LIN {X 0,Y 179.548,Z 284.993,A -85,B 0,C 180,E1 -23297.425,E2 -23297.425} C_VEL
LIN {X 0,Y 177.961,Z 297.46,A -85,B 0,C 180,E1 -23298.756,E2 -23298.756} C_VEL
LIN {X 0,Y 175.864,Z 309.48,A -85,B 0,C 180,E1 -23300.512,E2 -23300.512} C_VEL
LIN {X 0,Y 173.503,Z 321.02,A -85,B 0,C 180,E1 -23302.728,E2 -23302.728} C_VEL
LIN {X 0,Y 171.099,Z 331.401,A -85,B 0,C 180,E1 -23305.288,E2 -23305.288} C_VEL
LIN {X 0,Y 168.757,Z 340.608,A -85,B 0,C 180,E1 -23308.165,E2 -23308.165} C_VEL
LIN {X 0,Y 166.404,Z 349.816,A -85,B 0,C 180,E1 -23311.816,E2 -23311.816} C_VEL
LIN {X 0,Y 164.57,Z 357.07,A -85,B 0,C 180,E1 -23315.514,E2 -23315.514} C_VEL
LIN {X 0,Y 163.456,Z 361.84,A -85,B 0,C 180,E1 -23318.543,E2 -23318.543} C_VEL
LIN {X 0,Y 162.432,Z 366.745,A -85,B 0,C 180,E1 -23322.494,E2 -23322.494} C_VEL
LIN {X 0,Y 161.785,Z 370.877,A -85,B 0,C 180,E1 -23327.122,E2 -23327.122} C_VEL
LIN {X 0,Y 161.717,Z 372.885,A -85,B 0,C 180,E1 -23330.345,E2 -23330.345} C_VEL
LIN {X 0,Y 162.098,Z 374.429,A -85,B 0,C 180,E1 -23334.429,E2 -23334.429} C_VEL
LIN {X 0,Y 162.982,Z 374.928,A -85,B 0,C 180,E1 -23338.317,E2 -23338.317} C_VEL
LIN {X 0,Y 163.99,Z 374.684,A -85,B 0,C 180,E1 -23341.006,E2 -23341.006} C_VEL
LIN {X 0,Y 165.154,Z 374.032,A -85,B 0,C 180,E1 -23343.588,E2 -23343.588} C_VEL
LIN {X 0,Y 167.197,Z 372.422,A -85,B 0,C 180,E1 -23346.999,E2 -23346.999} C_VEL
LIN {X 0,Y 170.505,Z 369.157,A -85,B 0,C 180,E1 -23351.262,E2 -23351.262} C_VEL
LIN {X 0,Y 174.174,Z 364.95,A -85,B 0,C 180,E1 -23354.922,E2 -23354.922} C_VEL
LIN {X 0,Y 178.523,Z 359.365,A -85,B 0,C 180,E1 -23358.416,E2 -23358.416} C_VEL
LIN {X 0,Y 183.339,Z 352.372,A -85,B 0,C 180,E1 -23361.694,E2 -23361.694} C_VEL
LIN {X 0,Y 187.993,Z 344.807,A -85,B 0,C 180,E1 -23364.401,E2 -23364.401} C_VEL
LIN {X 0,Y 192.983,Z 335.71,A -85,B 0,C 180,E1 -23366.889,E2 -23366.889} C_VEL
LIN {X 0,Y 197.688,Z 325.505,A -85,B 0,C 180,E1 -23369.056,E2 -23369.056} C_VEL
LIN {X 0,Y 201.931,Z 314.615,A -85,B 0,C 180,E1 -23370.84,E2 -23370.84} C_VEL
LIN {X 0,Y 205.391,Z 303.558,A -85,B 0,C 180,E1 -23372.246,E2 -23372.246} C_VEL
LIN {X 0,Y 208.324,Z 291.535,A -85,B 0,C 180,E1 -23373.381,E2 -23373.381} C_VEL
LIN {X 0,Y 210.674,Z 278.298,A -85,B 0,C 180,E1 -23374.252,E2 -23374.252} C_VEL
LIN {X 0,Y 212.138,Z 264.43,A -85,B 0,C 180,E1 -23374.805,E2 -23374.805} C_VEL
LIN {X 0,Y 213.949,Z 239.049,A -85,B 0,C 180,E1 -23375.612,E2 -23375.612} C_VEL
LIN {X 0,Y 208.605,Z 229.191,A -85,B 0,C 180,E1 -23378.297,E2 -23378.297} C_VEL
LIN {X 0,Y 203.341,Z 220.675,A -85,B 0,C 180,E1 -23381.215,E2 -23381.215} C_VEL
LIN {X 0,Y 199.356,Z 214.616,A -85,B 0,C 180,E1 -23383.718,E2 -23383.718} C_VEL
LIN {X 0,Y 196.28,Z 210.234,A -85,B 0,C 180,E1 -23385.882,E2 -23385.882} C_VEL
LIN {X 0,Y 193.685,Z 206.523,A -85,B 0,C 180,E1 -23387.912,E2 -23387.912} C_VEL
LIN {X 0,Y 190.92,Z 202.867,A -85,B 0,C 180,E1 -23390.318,E2 -23390.318} C_VEL
LIN {X 0,Y 189.964,Z 201.478,A -85,B 0,C 180,E1 -23391.26,E2 -23391.26} C_VEL
LIN {X 0,Y 187.46,Z 198.302,A -85,B 0,C 180,E1 -23394.007,E2 -23394.007} C_VEL
LIN {X 0,Y 186.827,Z 196.888,A -85,B 0,C 180,E1 -23394.875,E2 -23394.875} C_VEL
LIN {X 0,Y 184.491,Z 195.131,A -85,B 0,C 180,E1 -23398.022,E2 -23398.022} C_VEL
LIN {X 0,Y 182.899,Z 191.675,A -85,B 0,C 180,E1 -23401.424,E2 -23401.424} C_VEL
LIN {X 0,Y 182.812,Z 191.257,A -85,B 0,C 180,E1 -23401.721,E2 -23401.721} C_VEL
LIN {X 0,Y 181.001,Z 190.735,A -85,B 0,C 180,E1 -23408.935,E2 -23408.935} C_VEL
LIN {X 0,Y 182.264,Z 191.532,A -85,B 0,C 180,E1 -23416.515,E2 -23416.515} C_VEL
LIN {X 0,Y 183.857,Z 194.886,A -85,B 0,C 180,E1 -23420.415,E2 -23420.415} C_VEL
LIN {X 0,Y 185.035,Z 196.289,A -85,B 0,C 180,E1 -23422.323,E2 -23422.323} C_VEL
LIN {X 0,Y 187.55,Z 199.714,A -85,B 0,C 180,E1 -23425.696,E2 -23425.696} C_VEL
LIN {X 0,Y 191.881,Z 206.408,A -85,B 0,C 180,E1 -23430.2,E2 -23430.2} C_VEL
LIN {X 0,Y 195.438,Z 212.282,A -85,B 0,C 180,E1 -23433.19,E2 -23433.19} C_VEL
LIN {X 0,Y 198.811,Z 218.156,A -85,B 0,C 180,E1 -23435.681,E2 -23435.681} C_VEL
LIN {X 0,Y 201.507,Z 223.122,A -85,B 0,C 180,E1 -23437.478,E2 -23437.478} C_VEL
LIN {X 0,Y 205.353,Z 230.604,A -85,B 0,C 180,E1 -23439.809,E2 -23439.809} C_VEL
LIN {X 0,Y 209.884,Z 240.49,A -85,B 0,C 180,E1 -23442.343,E2 -23442.343} C_VEL
LIN {X 0,Y 213.221,Z 249.266,A -85,B 0,C 180,E1 -23444.131,E2 -23444.131} C_VEL
LIN {X 0,Y 210.536,Z 285.028,A -85,B 0,C 180,E1 -23445.314,E2 -23445.314} C_VEL
LIN {X 0,Y 208.304,Z 298.59,A -85,B 0,C 180,E1 -23445.996,E2 -23445.996} C_VEL
LIN {X 0,Y 205.275,Z 311.214,A -85,B 0,C 180,E1 -23446.952,E2 -23446.952} C_VEL
LIN {X 0,Y 201.59,Z 322.873,A -85,B 0,C 180,E1 -23448.183,E2 -23448.183} C_VEL
LIN {X 0,Y 197.211,Z 334.157,A -85,B 0,C 180,E1 -23449.765,E2 -23449.765} C_VEL
LIN {X 0,Y 192.604,Z 344.363,A -85,B 0,C 180,E1 -23451.66,E2 -23451.66} C_VEL
LIN {X 0,Y 187.788,Z 353.573,A -85,B 0,C 180,E1 -23453.882,E2 -23453.882} C_VEL
LIN {X 0,Y 185.361,Z 357.845,A -85,B 0,C 180,E1 -23455.138,E2 -23455.138} C_VEL
LIN {X 0,Y 182.476,Z 361.648,A -85,B 0,C 180,E1 -23456.246,E2 -23456.246} C_VEL
LIN {X 0,Y 176.348,Z 367.396,A -85,B 0,C 180,E1 -23457.932,E2 -23457.932} C_VEL
LIN {X 0,Y 170.316,Z 372.485,A -85,B 0,C 180,E1 -23459.887,E2 -23459.887} C_VEL
LIN {X 0,Y 167.648,Z 375.204,A -85,B 0,C 180,E1 -23461.402,E2 -23461.402} C_VEL
LIN {X 0,Y 164.132,Z 379.67,A -85,B 0,C 180,E1 -23464.647,E2 -23464.647} C_VEL
LIN {X 0,Y 160.864,Z 383.343,A -85,B 0,C 180,E1 -23468.2,E2 -23468.2} C_VEL
LIN {X 0,Y 158.266,Z 386.042,A -85,B 0,C 180,E1 -23471.889,E2 -23471.889} C_VEL
LIN {X 0,Y 156.008,Z 388.264,A -85,B 0,C 180,E1 -23476.982,E2 -23476.982} C_VEL
LIN {X 0,Y 154.951,Z 388.886,A -85,B 0,C 180,E1 -23482.179,E2 -23482.179} C_VEL
LIN {X 0,Y 154.965,Z 388.002,A -85,B 0,C 180,E1 -23487.4,E2 -23487.4} C_VEL
LIN {X 0,Y 155.143,Z 386.944,A -85,B 0,C 180,E1 -23490,E2 -23490} C_VEL
LIN {X 0,Y 154.925,Z 384.718,A -85,B 0,C 180,E1 -23493.608,E2 -23493.608} C_VEL
LIN {X 0,Y 155.031,Z 381.017,A -85,B 0,C 180,E1 -23497.816,E2 -23497.816} C_VEL
LIN {X 0,Y 155.593,Z 376.389,A -85,B 0,C 180,E1 -23501.727,E2 -23501.727} C_VEL
LIN {X 0,Y 157.019,Z 369.344,A -85,B 0,C 180,E1 -23506.244,E2 -23506.244} C_VEL
LIN {X 0,Y 158.852,Z 361.682,A -85,B 0,C 180,E1 -23510.052,E2 -23510.052} C_VEL
LIN {X 0,Y 161.156,Z 352.661,A -85,B 0,C 180,E1 -23513.551,E2 -23513.551} C_VEL
LIN {X 0,Y 163.744,Z 343.153,A -85,B 0,C 180,E1 -23516.442,E2 -23516.442} C_VEL
LIN {X 0,Y 166.066,Z 333.554,A -85,B 0,C 180,E1 -23518.776,E2 -23518.776} C_VEL
LIN {X 0,Y 168.766,Z 321.638,A -85,B 0,C 180,E1 -23521.02,E2 -23521.02} C_VEL
LIN {X 0,Y 171.149,Z 308.858,A -85,B 0,C 180,E1 -23522.787,E2 -23522.787} C_VEL
LIN {X 0,Y 172.972,Z 296.083,A -85,B 0,C 180,E1 -23524.051,E2 -23524.051} C_VEL
LIN {X 0,Y 174.282,Z 282.642,A -85,B 0,C 180,E1 -23524.884,E2 -23524.884} C_VEL
LIN {X 0,Y 176.267,Z 240.088,A -85,B 0,C 180,E1 -23526.576,E2 -23526.576} C_VEL
LIN {X 0,Y 173.851,Z 214.223,A -85,B 0,C 180,E1 -23528.266,E2 -23528.266} C_VEL
LIN {X 0,Y 167.643,Z 197.165,A -85,B 0,C 180,E1 -23530.399,E2 -23530.399} C_VEL
LIN {X 0,Y 161.572,Z 183.654,A -85,B 0,C 180,E1 -23532.526,E2 -23532.526} C_VEL
LIN {X 0,Y 157.648,Z 175.577,A -85,B 0,C 180,E1 -23534.044,E2 -23534.044} C_VEL
LIN {X 0,Y 157.234,Z 173.902,A -85,B 0,C 180,E1 -23535.304,E2 -23535.304} C_VEL
LIN {X 0,Y 157.207,Z 173.906,A -85,B 0,C 180,E1 -23541.253,E2 -23541.253} C_VEL
LIN {X 0,Y 157.279,Z 173.895,A -85,B 0,C 180,E1 -23544.485,E2 -23544.485} C_VEL
LIN {X 0,Y 157.302,Z 173.892,A -85,B 0,C 180,E1 -23548.09,E2 -23548.09} C_VEL
LIN {X 0,Y 157.316,Z 173.889,A -85,B 0,C 180,E1 -23553.464,E2 -23553.464} C_VEL
LIN {X 0,Y 157.377,Z 173.846,A -85,B 0,C 180,E1 -23559.684,E2 -23559.684} C_VEL
LIN {X 0,Y 157.42,Z 173.84,A -85,B 0,C 180,E1 -23564.462,E2 -23564.462} C_VEL
LIN {X 0,Y 157.687,Z 173.84,A -85,B 0,C 180,E1 -23569.73,E2 -23569.73} C_VEL
LIN {X 0,Y 157.761,Z 173.82,A -85,B 0,C 180,E1 -23572.319,E2 -23572.319} C_VEL
LIN {X 0,Y 158.257,Z 173.763,A -85,B 0,C 180,E1 -23579.999,E2 -23579.999} C_VEL
LIN {X 0,Y 157.768,Z 173.828,A -85,B 0,C 180,E1 -23587.679,E2 -23587.679} C_VEL
LIN {X 0,Y 157.637,Z 173.828,A -85,B 0,C 180,E1 -23591.237,E2 -23591.237} C_VEL
LIN {X 0,Y 157.453,Z 173.87,A -85,B 0,C 180,E1 -23595.534,E2 -23595.534} C_VEL
LIN {X 0,Y 157.367,Z 173.863,A -85,B 0,C 180,E1 -23600.933,E2 -23600.933} C_VEL
LIN {X 0,Y 157.308,Z 173.888,A -85,B 0,C 180,E1 -23606.681,E2 -23606.681} C_VEL
LIN {X 0,Y 157.273,Z 173.885,A -85,B 0,C 180,E1 -23612.427,E2 -23612.427} C_VEL
LIN {X 0,Y 157.267,Z 173.886,A -85,B 0,C 180,E1 -23616.449,E2 -23616.449} C_VEL
LIN {X 0,Y 157.209,Z 173.899,A -85,B 0,C 180,E1 -23622.111,E2 -23622.111} C_VEL
LIN {X 0,Y 157.209,Z 173.9,A -85,B 0,C 180,E1 -23627.889,E2 -23627.889} C_VEL
LIN {X 0,Y 157.267,Z 173.895,A -85,B 0,C 180,E1 -23633.551,E2 -23633.551} C_VEL
LIN {X 0,Y 157.293,Z 173.868,A -85,B 0,C 180,E1 -23638.096,E2 -23638.096} C_VEL
LIN {X 0,Y 157.315,Z 173.887,A -85,B 0,C 180,E1 -23643.465,E2 -23643.465} C_VEL
LIN {X 0,Y 157.32,Z 173.875,A -85,B 0,C 180,E1 -23646.567,E2 -23646.567} C_VEL
LIN {X 0,Y 158.372,Z 176.829,A -85,B 0,C 180,E1 -23647.036,E2 -23647.036} C_VEL
LIN {X 0,Y 159.75,Z 178.723,A -85,B 0,C 180,E1 -23647.497,E2 -23647.497} C_VEL
LIN {X 0,Y 167.028,Z 191.548,A -85,B 0,C 180,E1 -23649.924,E2 -23649.924} C_VEL
LIN {X 0,Y 174.564,Z 207.153,A -85,B 0,C 180,E1 -23652.28,E2 -23652.28} C_VEL
LIN {X 0,Y 177.373,Z 213.874,A -85,B 0,C 180,E1 -23653.136,E2 -23653.136} C_VEL
LIN {X 0,Y 174.384,Z 271.947,A -85,B 0,C 180,E1 -23655.435,E2 -23655.435} C_VEL
LIN {X 0,Y 173.162,Z 285.336,A -85,B 0,C 180,E1 -23656.43,E2 -23656.43} C_VEL
LIN {X 0,Y 171.415,Z 298.31,A -85,B 0,C 180,E1 -23657.871,E2 -23657.871} C_VEL
LIN {X 0,Y 169.113,Z 311.003,A -85,B 0,C 180,E1 -23659.827,E2 -23659.827} C_VEL
LIN {X 0,Y 166.632,Z 322.332,A -85,B 0,C 180,E1 -23662.122,E2 -23662.122} C_VEL
LIN {X 0,Y 164.169,Z 332.474,A -85,B 0,C 180,E1 -23664.781,E2 -23664.781} C_VEL
LIN {X 0,Y 161.493,Z 342.364,A -85,B 0,C 180,E1 -23668.067,E2 -23668.067} C_VEL
LIN {X 0,Y 159.494,Z 349.969,A -85,B 0,C 180,E1 -23671.263,E2 -23671.263} C_VEL
LIN {X 0,Y 157.571,Z 357.268,A -85,B 0,C 180,E1 -23675.118,E2 -23675.118} C_VEL
LIN {X 0,Y 156.092,Z 363.349,A -85,B 0,C 180,E1 -23679.275,E2 -23679.275} C_VEL
LIN {X 0,Y 155.199,Z 367.652,A -85,B 0,C 180,E1 -23683.087,E2 -23683.087} C_VEL
LIN {X 0,Y 154.668,Z 371.258,A -85,B 0,C 180,E1 -23687.405,E2 -23687.405} C_VEL
LIN {X 0,Y 154.647,Z 373.49,A -85,B 0,C 180,E1 -23691.32,E2 -23691.32} C_VEL
LIN {X 0,Y 155.099,Z 374.767,A -85,B 0,C 180,E1 -23695.008,E2 -23695.008} C_VEL
LIN {X 0,Y 156.303,Z 375.234,A -85,B 0,C 180,E1 -23699.644,E2 -23699.644} C_VEL
LIN {X 0,Y 157.411,Z 374.925,A -85,B 0,C 180,E1 -23702.397,E2 -23702.397} C_VEL
LIN {X 0,Y 158.798,Z 374.161,A -85,B 0,C 180,E1 -23705.124,E2 -23705.124} C_VEL
LIN {X 0,Y 160.688,Z 372.749,A -85,B 0,C 180,E1 -23708.07,E2 -23708.07} C_VEL
LIN {X 0,Y 163.571,Z 370.108,A -85,B 0,C 180,E1 -23711.758,E2 -23711.758} C_VEL
LIN {X 0,Y 167.366,Z 366.135,A -85,B 0,C 180,E1 -23715.551,E2 -23715.551} C_VEL
LIN {X 0,Y 171.769,Z 360.946,A -85,B 0,C 180,E1 -23719.108,E2 -23719.108} C_VEL
LIN {X 0,Y 176.938,Z 354.011,A -85,B 0,C 180,E1 -23722.6,E2 -23722.6} C_VEL
LIN {X 0,Y 182.621,Z 345.319,A -85,B 0,C 180,E1 -23725.834,E2 -23725.834} C_VEL
LIN {X 0,Y 188.047,Z 335.855,A -85,B 0,C 180,E1 -23728.451,E2 -23728.451} C_VEL
LIN {X 0,Y 192.728,Z 326.162,A -85,B 0,C 180,E1 -23730.532,E2 -23730.532} C_VEL
LIN {X 0,Y 197.424,Z 314.624,A -85,B 0,C 180,E1 -23732.434,E2 -23732.434} C_VEL
LIN {X 0,Y 201.089,Z 303.238,A -85,B 0,C 180,E1 -23733.867,E2 -23733.867} C_VEL
LIN {X 0,Y 204.162,Z 290.943,A -85,B 0,C 180,E1 -23735.009,E2 -23735.009} C_VEL
LIN {X 0,Y 206.548,Z 277.661,A -85,B 0,C 180,E1 -23735.861,E2 -23735.861} C_VEL
LIN {X 0,Y 208.091,Z 262.604,A -85,B 0,C 180,E1 -23736.425,E2 -23736.425} C_VEL
LIN {X 0,Y 209.606,Z 242.189,A -85,B 0,C 180,E1 -23737.078,E2 -23737.078} C_VEL
LIN {X 0,Y 204.712,Z 233.173,A -85,B 0,C 180,E1 -23739.716,E2 -23739.716} C_VEL
LIN {X 0,Y 199.554,Z 224.573,A -85,B 0,C 180,E1 -23742.828,E2 -23742.828} C_VEL
LIN {X 0,Y 194.569,Z 216.973,A -85,B 0,C 180,E1 -23746.359,E2 -23746.359} C_VEL
LIN {X 0,Y 191.483,Z 212.642,A -85,B 0,C 180,E1 -23748.874,E2 -23748.874} C_VEL
LIN {X 0,Y 188.376,Z 208.146,A -85,B 0,C 180,E1 -23751.866,E2 -23751.866} C_VEL
LIN {X 0,Y 185.843,Z 204.684,A -85,B 0,C 180,E1 -23754.822,E2 -23754.822} C_VEL
LIN {X 0,Y 185.246,Z 203.644,A -85,B 0,C 180,E1 -23755.649,E2 -23755.649} C_VEL
LIN {X 0,Y 183.072,Z 201.682,A -85,B 0,C 180,E1 -23758.839,E2 -23758.839} C_VEL
LIN {X 0,Y 181.687,Z 198.253,A -85,B 0,C 180,E1 -23762.217,E2 -23762.217} C_VEL
LIN {X 0,Y 180.099,Z 197.78,A -85,B 0,C 180,E1 -23768.981,E2 -23768.981} C_VEL
LIN {X 0,Y 181.311,Z 198.564,A -85,B 0,C 180,E1 -23776.389,E2 -23776.389} C_VEL
LIN {X 0,Y 182.429,Z 201.419,A -85,B 0,C 180,E1 -23779.491,E2 -23779.491} C_VEL
LIN {X 0,Y 183.805,Z 203.167,A -85,B 0,C 180,E1 -23781.889,E2 -23781.889} C_VEL
LIN {X 0,Y 185.971,Z 206.206,A -85,B 0,C 180,E1 -23784.953,E2 -23784.953} C_VEL
LIN {X 0,Y 190.096,Z 212.929,A -85,B 0,C 180,E1 -23789.523,E2 -23789.523} C_VEL
LIN {X 0,Y 193.214,Z 218.303,A -85,B 0,C 180,E1 -23792.294,E2 -23792.294} C_VEL
LIN {X 0,Y 196.367,Z 224.046,A -85,B 0,C 180,E1 -23794.768,E2 -23794.768} C_VEL
LIN {X 0,Y 198.887,Z 228.945,A -85,B 0,C 180,E1 -23796.574,E2 -23796.574} C_VEL
LIN {X 0,Y 202.422,Z 236.118,A -85,B 0,C 180,E1 -23798.849,E2 -23798.849} C_VEL
LIN {X 0,Y 206.537,Z 245.513,A -85,B 0,C 180,E1 -23801.297,E2 -23801.297} C_VEL
LIN {X 0,Y 208.914,Z 251.869,A -85,B 0,C 180,E1 -23802.658,E2 -23802.658} C_VEL
LIN {X 0,Y 206.26,Z 284.992,A -85,B 0,C 180,E1 -23803.76,E2 -23803.76} C_VEL
LIN {X 0,Y 203.866,Z 298.863,A -85,B 0,C 180,E1 -23804.463,E2 -23804.463} C_VEL
LIN {X 0,Y 201.053,Z 310.175,A -85,B 0,C 180,E1 -23805.314,E2 -23805.314} C_VEL
LIN {X 0,Y 197.58,Z 321.095,A -85,B 0,C 180,E1 -23806.435,E2 -23806.435} C_VEL
LIN {X 0,Y 193.031,Z 332.621,A -85,B 0,C 180,E1 -23808.009,E2 -23808.009} C_VEL
LIN {X 0,Y 188.123,Z 343.034,A -85,B 0,C 180,E1 -23809.876,E2 -23809.876} C_VEL
LIN {X 0,Y 183.089,Z 352.461,A -85,B 0,C 180,E1 -23812.108,E2 -23812.108} C_VEL
LIN {X 0,Y 177.482,Z 361.58,A -85,B 0,C 180,E1 -23814.957,E2 -23814.957} C_VEL
LIN {X 0,Y 172.329,Z 368.965,A -85,B 0,C 180,E1 -23817.983,E2 -23817.983} C_VEL
LIN {X 0,Y 167.648,Z 375.204,A -85,B 0,C 180,E1 -23821.402,E2 -23821.402} C_VEL
LIN {X 0,Y 165.057,Z 377.763,A -85,B 0,C 180,E1 -23823.025,E2 -23823.025} C_VEL
LIN {X 0,Y 157.082,Z 382.585,A -85,B 0,C 180,E1 -23826.696,E2 -23826.696} C_VEL
LIN {X 0,Y 153.163,Z 384.683,A -85,B 0,C 180,E1 -23829.108,E2 -23829.108} C_VEL
LIN {X 0,Y 151.908,Z 385.532,A -85,B 0,C 180,E1 -23830.463,E2 -23830.463} C_VEL
LIN {X 0,Y 150.07,Z 387.165,A -85,B 0,C 180,E1 -23833.68,E2 -23833.68} C_VEL
LIN {X 0,Y 148.349,Z 388.459,A -85,B 0,C 180,E1 -23839.076,E2 -23839.076} C_VEL
LIN {X 0,Y 147.773,Z 388.244,A -85,B 0,C 180,E1 -23844.541,E2 -23844.541} C_VEL
LIN {X 0,Y 147.885,Z 387.559,A -85,B 0,C 180,E1 -23847.276,E2 -23847.276} C_VEL
LIN {X 0,Y 148.062,Z 386.428,A -85,B 0,C 180,E1 -23849.999,E2 -23849.999} C_VEL
LIN {X 0,Y 147.843,Z 384.435,A -85,B 0,C 180,E1 -23853.354,E2 -23853.354} C_VEL
LIN {X 0,Y 147.981,Z 380.32,A -85,B 0,C 180,E1 -23858.191,E2 -23858.191} C_VEL
LIN {X 0,Y 148.6,Z 375.582,A -85,B 0,C 180,E1 -23862.288,E2 -23862.288} C_VEL
LIN {X 0,Y 150.157,Z 368.421,A -85,B 0,C 180,E1 -23867.009,E2 -23867.009} C_VEL
LIN {X 0,Y 152.156,Z 360.601,A -85,B 0,C 180,E1 -23870.975,E2 -23870.975} C_VEL
LIN {X 0,Y 154.299,Z 352.561,A -85,B 0,C 180,E1 -23874.2,E2 -23874.2} C_VEL
LIN {X 0,Y 156.796,Z 343.857,A -85,B 0,C 180,E1 -23876.989,E2 -23876.989} C_VEL
LIN {X 0,Y 159.487,Z 333.154,A -85,B 0,C 180,E1 -23879.718,E2 -23879.718} C_VEL
LIN {X 0,Y 162.313,Z 321.215,A -85,B 0,C 180,E1 -23882.033,E2 -23882.033} C_VEL
LIN {X 0,Y 164.791,Z 308.406,A -85,B 0,C 180,E1 -23883.854,E2 -23883.854} C_VEL
LIN {X 0,Y 166.665,Z 295.567,A -85,B 0,C 180,E1 -23885.16,E2 -23885.16} C_VEL
LIN {X 0,Y 168.055,Z 281.84,A -85,B 0,C 180,E1 -23886.016,E2 -23886.016} C_VEL
LIN {X 0,Y 170.072,Z 240.808,A -85,B 0,C 180,E1 -23887.69,E2 -23887.69} C_VEL
LIN {X 0,Y 167.799,Z 216.274,A -85,B 0,C 180,E1 -23889.382,E2 -23889.382} C_VEL
LIN {X 0,Y 162.112,Z 200.421,A -85,B 0,C 180,E1 -23891.479,E2 -23891.479} C_VEL
LIN {X 0,Y 156.28,Z 187.267,A -85,B 0,C 180,E1 -23893.661,E2 -23893.661} C_VEL
LIN {X 0,Y 151.543,Z 178.113,A -85,B 0,C 180,E1 -23895.492,E2 -23895.492} C_VEL
LIN {X 0,Y 150.326,Z 175.58,A -85,B 0,C 180,E1 -23895.999,E2 -23895.999} C_VEL
LIN {X 0,Y 150.138,Z 174.786,A -85,B 0,C 180,E1 -23896.456,E2 -23896.456} C_VEL
LIN {X 0,Y 150.173,Z 174.782,A -85,B 0,C 180,E1 -23902.526,E2 -23902.526} C_VEL
LIN {X 0,Y 150.221,Z 174.774,A -85,B 0,C 180,E1 -23907.364,E2 -23907.364} C_VEL
LIN {X 0,Y 150.242,Z 174.77,A -85,B 0,C 180,E1 -23912.719,E2 -23912.719} C_VEL
LIN {X 0,Y 150.339,Z 174.727,A -85,B 0,C 180,E1 -23919.219,E2 -23919.219} C_VEL
LIN {X 0,Y 150.327,Z 174.712,A -85,B 0,C 180,E1 -23923.709,E2 -23923.709} C_VEL
LIN {X 0,Y 150.607,Z 174.723,A -85,B 0,C 180,E1 -23929.242,E2 -23929.242} C_VEL
LIN {X 0,Y 150.699,Z 174.702,A -85,B 0,C 180,E1 -23931.957,E2 -23931.957} C_VEL
LIN {X 0,Y 151.217,Z 174.639,A -85,B 0,C 180,E1 -23939.999,E2 -23939.999} C_VEL
LIN {X 0,Y 150.705,Z 174.708,A -85,B 0,C 180,E1 -23948.042,E2 -23948.042} C_VEL
LIN {X 0,Y 150.577,Z 174.706,A -85,B 0,C 180,E1 -23951.437,E2 -23951.437} C_VEL
LIN {X 0,Y 150.361,Z 174.755,A -85,B 0,C 180,E1 -23956.286,E2 -23956.286} C_VEL
LIN {X 0,Y 150.348,Z 174.736,A -85,B 0,C 180,E1 -23960.79,E2 -23960.79} C_VEL
LIN {X 0,Y 150.24,Z 174.768,A -85,B 0,C 180,E1 -23967.279,E2 -23967.279} C_VEL
LIN {X 0,Y 150.213,Z 174.765,A -85,B 0,C 180,E1 -23972.632,E2 -23972.632} C_VEL
LIN {X 0,Y 150.171,Z 174.763,A -85,B 0,C 180,E1 -23977.473,E2 -23977.473} C_VEL
LIN {X 0,Y 150.149,Z 174.778,A -85,B 0,C 180,E1 -23981.505,E2 -23981.505} C_VEL
LIN {X 0,Y 150.123,Z 174.771,A -85,B 0,C 180,E1 -23985.395,E2 -23985.395} C_VEL
LIN {X 0,Y 150.15,Z 174.781,A -85,B 0,C 180,E1 -23989.059,E2 -23989.059} C_VEL
LIN {X 0,Y 150.178,Z 174.774,A -85,B 0,C 180,E1 -23992.708,E2 -23992.708} C_VEL
LIN {X 0,Y 150.214,Z 174.752,A -85,B 0,C 180,E1 -23997.368,E2 -23997.368} C_VEL
LIN {X 0,Y 150.28,Z 174.762,A -85,B 0,C 180,E1 -24003.677,E2 -24003.677} C_VEL
LIN {X 0,Y 150.24,Z 174.758,A -85,B 0,C 180,E1 -24004.665,E2 -24004.665} C_VEL
LIN {X 0,Y 151.14,Z 177.478,A -85,B 0,C 180,E1 -24005.104,E2 -24005.104} C_VEL
LIN {X 0,Y 152.861,Z 179.883,A -85,B 0,C 180,E1 -24005.738,E2 -24005.738} C_VEL
LIN {X 0,Y 160.508,Z 192.897,A -85,B 0,C 180,E1 -24008.473,E2 -24008.473} C_VEL
LIN {X 0,Y 168.176,Z 208.642,A -85,B 0,C 180,E1 -24011.057,E2 -24011.057} C_VEL
LIN {X 0,Y 171.175,Z 215.566,A -85,B 0,C 180,E1 -24012.024,E2 -24012.024} C_VEL
LIN {X 0,Y 168.18,Z 271.347,A -85,B 0,C 180,E1 -24014.275,E2 -24014.275} C_VEL
LIN {X 0,Y 166.908,Z 284.834,A -85,B 0,C 180,E1 -24015.278,E2 -24015.278} C_VEL
LIN {X 0,Y 165.281,Z 297.014,A -85,B 0,C 180,E1 -24016.632,E2 -24016.632} C_VEL
LIN {X 0,Y 162.991,Z 309.339,A -85,B 0,C 180,E1 -24018.497,E2 -24018.497} C_VEL
LIN {X 0,Y 160.413,Z 321.018,A -85,B 0,C 180,E1 -24020.862,E2 -24020.862} C_VEL
LIN {X 0,Y 157.778,Z 331.54,A -85,B 0,C 180,E1 -24023.607,E2 -24023.607} C_VEL
LIN {X 0,Y 155.09,Z 341.162,A -85,B 0,C 180,E1 -24026.825,E2 -24026.825} C_VEL
LIN {X 0,Y 152.603,Z 350.122,A -85,B 0,C 180,E1 -24030.66,E2 -24030.66} C_VEL
LIN {X 0,Y 150.596,Z 357.463,A -85,B 0,C 180,E1 -24034.685,E2 -24034.685} C_VEL
LIN {X 0,Y 148.934,Z 363.98,A -85,B 0,C 180,E1 -24039.37,E2 -24039.37} C_VEL
LIN {X 0,Y 147.989,Z 368.559,A -85,B 0,C 180,E1 -24043.737,E2 -24043.737} C_VEL
LIN {X 0,Y 147.544,Z 371.629,A -85,B 0,C 180,E1 -24047.701,E2 -24047.701} C_VEL
LIN {X 0,Y 147.621,Z 374.097,A -85,B 0,C 180,E1 -24052.388,E2 -24052.388} C_VEL
LIN {X 0,Y 148.12,Z 375.106,A -85,B 0,C 180,E1 -24055.644,E2 -24055.644} C_VEL
LIN {X 0,Y 149.71,Z 375.541,A -85,B 0,C 180,E1 -24061.091,E2 -24061.091} C_VEL
LIN {X 0,Y 150.972,Z 375.141,A -85,B 0,C 180,E1 -24063.961,E2 -24063.961} C_VEL
LIN {X 0,Y 154.224,Z 373.081,A -85,B 0,C 180,E1 -24069.224,E2 -24069.224} C_VEL
LIN {X 0,Y 157.874,Z 369.944,A -85,B 0,C 180,E1 -24073.631,E2 -24073.631} C_VEL
LIN {X 0,Y 162.039,Z 365.792,A -85,B 0,C 180,E1 -24077.505,E2 -24077.505} C_VEL
LIN {X 0,Y 167.169,Z 359.938,A -85,B 0,C 180,E1 -24081.357,E2 -24081.357} C_VEL
LIN {X 0,Y 172.365,Z 353.202,A -85,B 0,C 180,E1 -24084.636,E2 -24084.636} C_VEL
LIN {X 0,Y 177.368,Z 345.881,A -85,B 0,C 180,E1 -24087.353,E2 -24087.353} C_VEL
LIN {X 0,Y 182.714,Z 337.094,A -85,B 0,C 180,E1 -24089.847,E2 -24089.847} C_VEL
LIN {X 0,Y 187.906,Z 326.882,A -85,B 0,C 180,E1 -24092.082,E2 -24092.082} C_VEL
LIN {X 0,Y 192.356,Z 316.541,A -85,B 0,C 180,E1 -24093.818,E2 -24093.818} C_VEL
LIN {X 0,Y 196.277,Z 305.22,A -85,B 0,C 180,E1 -24095.312,E2 -24095.312} C_VEL
LIN {X 0,Y 199.383,Z 293.936,A -85,B 0,C 180,E1 -24096.416,E2 -24096.416} C_VEL
LIN {X 0,Y 201.918,Z 281.357,A -85,B 0,C 180,E1 -24097.287,E2 -24097.287} C_VEL
LIN {X 0,Y 203.591,Z 268.319,A -85,B 0,C 180,E1 -24097.869,E2 -24097.869} C_VEL
LIN {X 0,Y 205.426,Z 245.497,A -85,B 0,C 180,E1 -24098.586,E2 -24098.586} C_VEL
LIN {X 0,Y 200.659,Z 236.654,A -85,B 0,C 180,E1 -24101.366,E2 -24101.366} C_VEL
LIN {X 0,Y 195.929,Z 228.633,A -85,B 0,C 180,E1 -24104.521,E2 -24104.521} C_VEL
LIN {X 0,Y 191.884,Z 222.435,A -85,B 0,C 180,E1 -24107.628,E2 -24107.628} C_VEL
LIN {X 0,Y 189.706,Z 219.161,A -85,B 0,C 180,E1 -24109.529,E2 -24109.529} C_VEL
LIN {X 0,Y 186.624,Z 214.55,A -85,B 0,C 180,E1 -24112.689,E2 -24112.689} C_VEL
LIN {X 0,Y 184.281,Z 211.104,A -85,B 0,C 180,E1 -24115.626,E2 -24115.626} C_VEL
LIN {X 0,Y 184.015,Z 210.524,A -85,B 0,C 180,E1 -24116.031,E2 -24116.031} C_VEL
LIN {X 0,Y 181.864,Z 208.482,A -85,B 0,C 180,E1 -24119.338,E2 -24119.338} C_VEL
LIN {X 0,Y 180.598,Z 205.274,A -85,B 0,C 180,E1 -24122.661,E2 -24122.661} C_VEL
LIN {X 0,Y 179.198,Z 204.826,A -85,B 0,C 180,E1 -24129.026,E2 -24129.026} C_VEL
LIN {X 0,Y 180.258,Z 205.526,A -85,B 0,C 180,E1 -24135.962,E2 -24135.962} C_VEL
LIN {X 0,Y 181.399,Z 208.427,A -85,B 0,C 180,E1 -24139.286,E2 -24139.286} C_VEL
LIN {X 0,Y 182.669,Z 210.167,A -85,B 0,C 180,E1 -24141.587,E2 -24141.587} C_VEL
LIN {X 0,Y 184.511,Z 212.919,A -85,B 0,C 180,E1 -24144.328,E2 -24144.328} C_VEL
LIN {X 0,Y 188.225,Z 219.264,A -85,B 0,C 180,E1 -24148.721,E2 -24148.721} C_VEL
LIN {X 0,Y 191.063,Z 224.415,A -85,B 0,C 180,E1 -24151.405,E2 -24151.405} C_VEL
LIN {X 0,Y 194.088,Z 230.158,A -85,B 0,C 180,E1 -24153.922,E2 -24153.922} C_VEL
LIN {X 0,Y 197.593,Z 237.255,A -85,B 0,C 180,E1 -24156.527,E2 -24156.527} C_VEL
LIN {X 0,Y 202.024,Z 247.36,A -85,B 0,C 180,E1 -24159.445,E2 -24159.445} C_VEL
LIN {X 0,Y 204.714,Z 254.532,A -85,B 0,C 180,E1 -24161.111,E2 -24161.111} C_VEL
LIN {X 0,Y 202.214,Z 284.596,A -85,B 0,C 180,E1 -24162.127,E2 -24162.127} C_VEL
LIN {X 0,Y 199.872,Z 297.801,A -85,B 0,C 180,E1 -24162.775,E2 -24162.775} C_VEL
LIN {X 0,Y 196.776,Z 309.991,A -85,B 0,C 180,E1 -24163.677,E2 -24163.677} C_VEL
LIN {X 0,Y 193.149,Z 320.971,A -85,B 0,C 180,E1 -24164.802,E2 -24164.802} C_VEL
LIN {X 0,Y 188.446,Z 332.459,A -85,B 0,C 180,E1 -24166.373,E2 -24166.373} C_VEL
LIN {X 0,Y 183.364,Z 342.84,A -85,B 0,C 180,E1 -24168.244,E2 -24168.244} C_VEL
LIN {X 0,Y 178.613,Z 351.348,A -85,B 0,C 180,E1 -24170.252,E2 -24170.252} C_VEL
LIN {X 0,Y 173.652,Z 359.227,A -85,B 0,C 180,E1 -24172.621,E2 -24172.621} C_VEL
LIN {X 0,Y 168.08,Z 366.993,A -85,B 0,C 180,E1 -24175.633,E2 -24175.633} C_VEL
LIN {X 0,Y 163.126,Z 373.253,A -85,B 0,C 180,E1 -24178.868,E2 -24178.868} C_VEL
LIN {X 0,Y 158.979,Z 378.268,A -85,B 0,C 180,E1 -24182.333,E2 -24182.333} C_VEL
LIN {X 0,Y 155.332,Z 382.211,A -85,B 0,C 180,E1 -24185.97,E2 -24185.97} C_VEL
LIN {X 0,Y 151.908,Z 385.532,A -85,B 0,C 180,E1 -24190.463,E2 -24190.463} C_VEL
LIN {X 0,Y 150.006,Z 386.705,A -85,B 0,C 180,E1 -24192.54,E2 -24192.54} C_VEL
LIN {X 0,Y 145.636,Z 387.91,A -85,B 0,C 180,E1 -24195.96,E2 -24195.96} C_VEL
LIN {X 0,Y 142.417,Z 388.264,A -85,B 0,C 180,E1 -24198.849,E2 -24198.849} C_VEL
LIN {X 0,Y 140.987,Z 388.203,A -85,B 0,C 180,E1 -24201.173,E2 -24201.173} C_VEL
LIN {X 0,Y 140.814,Z 388.123,A -85,B 0,C 180,E1 -24201.971,E2 -24201.971} C_VEL
LIN {X 0,Y 140.806,Z 387.088,A -85,B 0,C 180,E1 -24207.138,E2 -24207.138} C_VEL
LIN {X 0,Y 140.984,Z 385.913,A -85,B 0,C 180,E1 -24209.999,E2 -24209.999} C_VEL
LIN {X 0,Y 140.779,Z 384.087,A -85,B 0,C 180,E1 -24213.183,E2 -24213.183} C_VEL
LIN {X 0,Y 140.817,Z 380.967,A -85,B 0,C 180,E1 -24217.167,E2 -24217.167} C_VEL
LIN {X 0,Y 141.345,Z 376.531,A -85,B 0,C 180,E1 -24221.471,E2 -24221.471} C_VEL
LIN {X 0,Y 142.471,Z 370.853,A -85,B 0,C 180,E1 -24225.742,E2 -24225.742} C_VEL
LIN {X 0,Y 144.37,Z 363.723,A -85,B 0,C 180,E1 -24229.923,E2 -24229.923} C_VEL
LIN {X 0,Y 146.542,Z 355.277,A -85,B 0,C 180,E1 -24233.809,E2 -24233.809} C_VEL
LIN {X 0,Y 149.543,Z 345.781,A -85,B 0,C 180,E1 -24237.196,E2 -24237.196} C_VEL
LIN {X 0,Y 152.068,Z 336.638,A -85,B 0,C 180,E1 -24239.79,E2 -24239.79} C_VEL
LIN {X 0,Y 154,Z 328.586,A -85,B 0,C 180,E1 -24241.655,E2 -24241.655} C_VEL
LIN {X 0,Y 156.681,Z 317.228,A -85,B 0,C 180,E1 -24243.716,E2 -24243.716} C_VEL
LIN {X 0,Y 158.946,Z 305.67,A -85,B 0,C 180,E1 -24245.28,E2 -24245.28} C_VEL
LIN {X 0,Y 160.774,Z 292.357,A -85,B 0,C 180,E1 -24246.555,E2 -24246.555} C_VEL
LIN {X 0,Y 161.977,Z 279.604,A -85,B 0,C 180,E1 -24247.306,E2 -24247.306} C_VEL
LIN {X 0,Y 163.916,Z 240.809,A -85,B 0,C 180,E1 -24248.932,E2 -24248.932} C_VEL
LIN {X 0,Y 161.817,Z 218.225,A -85,B 0,C 180,E1 -24250.586,E2 -24250.586} C_VEL
LIN {X 0,Y 156.535,Z 203.265,A -85,B 0,C 180,E1 -24252.686,E2 -24252.686} C_VEL
LIN {X 0,Y 150.1,Z 188.776,A -85,B 0,C 180,E1 -24255.263,E2 -24255.263} C_VEL
LIN {X 0,Y 145.544,Z 180.196,A -85,B 0,C 180,E1 -24257.173,E2 -24257.173} C_VEL
LIN {X 0,Y 143.728,Z 177.829,A -85,B 0,C 180,E1 -24257.913,E2 -24257.913} C_VEL
LIN {X 0,Y 143.109,Z 175.662,A -85,B 0,C 180,E1 -24258.358,E2 -24258.358} C_VEL
LIN {X 0,Y 143.088,Z 175.665,A -85,B 0,C 180,E1 -24263.885,E2 -24263.885} C_VEL
LIN {X 0,Y 143.187,Z 175.65,A -85,B 0,C 180,E1 -24267.322,E2 -24267.322} C_VEL
LIN {X 0,Y 143.19,Z 175.649,A -85,B 0,C 180,E1 -24272.062,E2 -24272.062} C_VEL
LIN {X 0,Y 143.267,Z 175.613,A -85,B 0,C 180,E1 -24278.755,E2 -24278.755} C_VEL
LIN {X 0,Y 143.266,Z 175.584,A -85,B 0,C 180,E1 -24282.882,E2 -24282.882} C_VEL
LIN {X 0,Y 143.533,Z 175.602,A -85,B 0,C 180,E1 -24288.705,E2 -24288.705} C_VEL
LIN {X 0,Y 143.621,Z 175.586,A -85,B 0,C 180,E1 -24291.558,E2 -24291.558} C_VEL
LIN {X 0,Y 144.175,Z 175.515,A -85,B 0,C 180,E1 -24299.999,E2 -24299.999} C_VEL
LIN {X 0,Y 143.626,Z 175.587,A -85,B 0,C 180,E1 -24308.441,E2 -24308.441} C_VEL
LIN {X 0,Y 143.505,Z 175.586,A -85,B 0,C 180,E1 -24311.63,E2 -24311.63} C_VEL
LIN {X 0,Y 143.301,Z 175.633,A -85,B 0,C 180,E1 -24317.113,E2 -24317.113} C_VEL
LIN {X 0,Y 143.274,Z 175.617,A -85,B 0,C 180,E1 -24321.252,E2 -24321.252} C_VEL
LIN {X 0,Y 143.187,Z 175.641,A -85,B 0,C 180,E1 -24327.935,E2 -24327.935} C_VEL
LIN {X 0,Y 143.142,Z 175.649,A -85,B 0,C 180,E1 -24333.42,E2 -24333.42} C_VEL
LIN {X 0,Y 143.06,Z 175.651,A -85,B 0,C 180,E1 -24339.69,E2 -24339.69} C_VEL
LIN {X 0,Y 143.054,Z 175.659,A -85,B 0,C 180,E1 -24343.455,E2 -24343.455} C_VEL
LIN {X 0,Y 143.063,Z 175.659,A -85,B 0,C 180,E1 -24347.465,E2 -24347.465} C_VEL
LIN {X 0,Y 143.076,Z 175.654,A -85,B 0,C 180,E1 -24351.806,E2 -24351.806} C_VEL
LIN {X 0,Y 143.181,Z 175.628,A -85,B 0,C 180,E1 -24357.322,E2 -24357.322} C_VEL
LIN {X 0,Y 143.21,Z 175.648,A -85,B 0,C 180,E1 -24362.508,E2 -24362.508} C_VEL
LIN {X 0,Y 144.199,Z 178.435,A -85,B 0,C 180,E1 -24363.037,E2 -24363.037} C_VEL
LIN {X 0,Y 145.798,Z 180.587,A -85,B 0,C 180,E1 -24363.689,E2 -24363.689} C_VEL
LIN {X 0,Y 154.137,Z 194.536,A -85,B 0,C 180,E1 -24366.949,E2 -24366.949} C_VEL
LIN {X 0,Y 161.116,Z 208.603,A -85,B 0,C 180,E1 -24369.479,E2 -24369.479} C_VEL
LIN {X 0,Y 165.112,Z 217.978,A -85,B 0,C 180,E1 -24370.882,E2 -24370.882} C_VEL
LIN {X 0,Y 161.931,Z 272.179,A -85,B 0,C 180,E1 -24373.118,E2 -24373.118} C_VEL
LIN {X 0,Y 160.574,Z 286.017,A -85,B 0,C 180,E1 -24374.206,E2 -24374.206} C_VEL
LIN {X 0,Y 158.674,Z 298.968,A -85,B 0,C 180,E1 -24375.737,E2 -24375.737} C_VEL
LIN {X 0,Y 156.316,Z 310.863,A -85,B 0,C 180,E1 -24377.669,E2 -24377.669} C_VEL
LIN {X 0,Y 153.599,Z 322.341,A -85,B 0,C 180,E1 -24380.121,E2 -24380.121} C_VEL
LIN {X 0,Y 150.882,Z 332.631,A -85,B 0,C 180,E1 -24382.977,E2 -24382.977} C_VEL
LIN {X 0,Y 148.139,Z 341.913,A -85,B 0,C 180,E1 -24386.251,E2 -24386.251} C_VEL
LIN {X 0,Y 145.739,Z 350.274,A -85,B 0,C 180,E1 -24390.001,E2 -24390.001} C_VEL
LIN {X 0,Y 143.62,Z 357.658,A -85,B 0,C 180,E1 -24394.21,E2 -24394.21} C_VEL
LIN {X 0,Y 142.046,Z 363.528,A -85,B 0,C 180,E1 -24398.537,E2 -24398.537} C_VEL
LIN {X 0,Y 141.019,Z 368.148,A -85,B 0,C 180,E1 -24402.96,E2 -24402.96} C_VEL
LIN {X 0,Y 140.435,Z 372.009,A -85,B 0,C 180,E1 -24408.04,E2 -24408.04} C_VEL
LIN {X 0,Y 140.668,Z 374.687,A -85,B 0,C 180,E1 -24413.56,E2 -24413.56} C_VEL
LIN {X 0,Y 141.201,Z 375.495,A -85,B 0,C 180,E1 -24416.613,E2 -24416.613} C_VEL
LIN {X 0,Y 142.029,Z 375.885,A -85,B 0,C 180,E1 -24419.659,E2 -24419.659} C_VEL
LIN {X 0,Y 143.635,Z 375.687,A -85,B 0,C 180,E1 -24423.717,E2 -24423.717} C_VEL
LIN {X 0,Y 146.459,Z 374.318,A -85,B 0,C 180,E1 -24428.596,E2 -24428.596} C_VEL
LIN {X 0,Y 148.593,Z 372.881,A -85,B 0,C 180,E1 -24431.465,E2 -24431.465} C_VEL
LIN {X 0,Y 152.157,Z 369.948,A -85,B 0,C 180,E1 -24435.434,E2 -24435.434} C_VEL
LIN {X 0,Y 156.931,Z 365.405,A -85,B 0,C 180,E1 -24439.582,E2 -24439.582} C_VEL
LIN {X 0,Y 162.005,Z 359.911,A -85,B 0,C 180,E1 -24443.168,E2 -24443.168} C_VEL
LIN {X 0,Y 168.027,Z 352.42,A -85,B 0,C 180,E1 -24446.777,E2 -24446.777} C_VEL
LIN {X 0,Y 173.356,Z 344.84,A -85,B 0,C 180,E1 -24449.485,E2 -24449.485} C_VEL
LIN {X 0,Y 178.655,Z 336.257,A -85,B 0,C 180,E1 -24451.832,E2 -24451.832} C_VEL
LIN {X 0,Y 183.847,Z 326.351,A -85,B 0,C 180,E1 -24453.942,E2 -24453.942} C_VEL
LIN {X 0,Y 188.852,Z 314.807,A -85,B 0,C 180,E1 -24455.836,E2 -24455.836} C_VEL
LIN {X 0,Y 192.878,Z 303.098,A -85,B 0,C 180,E1 -24457.269,E2 -24457.269} C_VEL
LIN {X 0,Y 196.094,Z 290.94,A -85,B 0,C 180,E1 -24458.373,E2 -24458.373} C_VEL
LIN {X 0,Y 198.484,Z 278.411,A -85,B 0,C 180,E1 -24459.162,E2 -24459.162} C_VEL
LIN {X 0,Y 200.122,Z 263.814,A -85,B 0,C 180,E1 -24459.703,E2 -24459.703} C_VEL
LIN {X 0,Y 201.29,Z 248.663,A -85,B 0,C 180,E1 -24460.214,E2 -24460.214} C_VEL
LIN {X 0,Y 196.492,Z 239.611,A -85,B 0,C 180,E1 -24463.307,E2 -24463.307} C_VEL
LIN {X 0,Y 192.079,Z 232.199,A -85,B 0,C 180,E1 -24466.582,E2 -24466.582} C_VEL
LIN {X 0,Y 188.32,Z 226.111,A -85,B 0,C 180,E1 -24469.861,E2 -24469.861} C_VEL
LIN {X 0,Y 184.964,Z 221.082,A -85,B 0,C 180,E1 -24473.455,E2 -24473.455} C_VEL
LIN {X 0,Y 182.484,Z 217.27,A -85,B 0,C 180,E1 -24476.827,E2 -24476.827} C_VEL
LIN {X 0,Y 180.497,Z 214.969,A -85,B 0,C 180,E1 -24480.236,E2 -24480.236} C_VEL
LIN {X 0,Y 179.524,Z 212.294,A -85,B 0,C 180,E1 -24483.095,E2 -24483.095} C_VEL
LIN {X 0,Y 178.284,Z 211.881,A -85,B 0,C 180,E1 -24489.764,E2 -24489.764} C_VEL
LIN {X 0,Y 179.231,Z 212.559,A -85,B 0,C 180,E1 -24495.606,E2 -24495.606} C_VEL
LIN {X 0,Y 180.443,Z 215.561,A -85,B 0,C 180,E1 -24499.232,E2 -24499.232} C_VEL
LIN {X 0,Y 181.535,Z 217.185,A -85,B 0,C 180,E1 -24501.282,E2 -24501.282} C_VEL
LIN {X 0,Y 183.068,Z 219.584,A -85,B 0,C 180,E1 -24503.681,E2 -24503.681} C_VEL
LIN {X 0,Y 186.363,Z 225.529,A -85,B 0,C 180,E1 -24507.856,E2 -24507.856} C_VEL
LIN {X 0,Y 189.027,Z 230.626,A -85,B 0,C 180,E1 -24510.558,E2 -24510.558} C_VEL
LIN {X 0,Y 192.053,Z 236.635,A -85,B 0,C 180,E1 -24513.218,E2 -24513.218} C_VEL
LIN {X 0,Y 196.054,Z 245.386,A -85,B 0,C 180,E1 -24516.331,E2 -24516.331} C_VEL
LIN {X 0,Y 199.97,Z 255.22,A -85,B 0,C 180,E1 -24519.038,E2 -24519.038} C_VEL
LIN {X 0,Y 200.702,Z 257.55,A -85,B 0,C 180,E1 -24519.541,E2 -24519.541} C_VEL
LIN {X 0,Y 198.316,Z 284.296,A -85,B 0,C 180,E1 -24520.428,E2 -24520.428} C_VEL
LIN {X 0,Y 195.814,Z 297.868,A -85,B 0,C 180,E1 -24521.086,E2 -24521.086} C_VEL
LIN {X 0,Y 192.633,Z 309.929,A -85,B 0,C 180,E1 -24521.981,E2 -24521.981} C_VEL
LIN {X 0,Y 188.884,Z 320.847,A -85,B 0,C 180,E1 -24523.095,E2 -24523.095} C_VEL
LIN {X 0,Y 184.022,Z 332.297,A -85,B 0,C 180,E1 -24524.658,E2 -24524.658} C_VEL
LIN {X 0,Y 178.713,Z 342.657,A -85,B 0,C 180,E1 -24526.512,E2 -24526.512} C_VEL
LIN {X 0,Y 173.243,Z 352.008,A -85,B 0,C 180,E1 -24528.759,E2 -24528.759} C_VEL
LIN {X 0,Y 167.073,Z 361.07,A -85,B 0,C 180,E1 -24531.649,E2 -24531.649} C_VEL
LIN {X 0,Y 161.367,Z 368.414,A -85,B 0,C 180,E1 -24534.754,E2 -24534.754} C_VEL
LIN {X 0,Y 155.539,Z 375.217,A -85,B 0,C 180,E1 -24538.692,E2 -24538.692} C_VEL
LIN {X 0,Y 151.383,Z 379.752,A -85,B 0,C 180,E1 -24542.338,E2 -24542.338} C_VEL
LIN {X 0,Y 146.684,Z 384.168,A -85,B 0,C 180,E1 -24547.461,E2 -24547.461} C_VEL
LIN {X 0,Y 144.802,Z 385.772,A -85,B 0,C 180,E1 -24550.138,E2 -24550.138} C_VEL
LIN {X 0,Y 143.237,Z 386.959,A -85,B 0,C 180,E1 -24552.878,E2 -24552.878} C_VEL
LIN {X 0,Y 141.36,Z 388.154,A -85,B 0,C 180,E1 -24558.529,E2 -24558.529} C_VEL
LIN {X 0,Y 140.814,Z 388.123,A -85,B 0,C 180,E1 -24561.971,E2 -24561.971} C_VEL
LIN {X 0,Y 139.988,Z 387.785,A -85,B 0,C 180,E1 -24564.358,E2 -24564.358} C_VEL
LIN {X 0,Y 138.374,Z 387.065,A -85,B 0,C 180,E1 -24566.703,E2 -24566.703} C_VEL
LIN {X 0,Y 134.763,Z 384.746,A -85,B 0,C 180,E1 -24571.437,E2 -24571.437} C_VEL
LIN {X 0,Y 133.682,Z 382.553,A -85,B 0,C 180,E1 -24574.705,E2 -24574.705} C_VEL
LIN {X 0,Y 133.899,Z 378.913,A -85,B 0,C 180,E1 -24579.059,E2 -24579.059} C_VEL
LIN {X 0,Y 134.699,Z 373.968,A -85,B 0,C 180,E1 -24583.579,E2 -24583.579} C_VEL
LIN {X 0,Y 136.211,Z 367.711,A -85,B 0,C 180,E1 -24588.033,E2 -24588.033} C_VEL
LIN {X 0,Y 138.429,Z 359.87,A -85,B 0,C 180,E1 -24592.381,E2 -24592.381} C_VEL
LIN {X 0,Y 140.666,Z 352.213,A -85,B 0,C 180,E1 -24595.746,E2 -24595.746} C_VEL
LIN {X 0,Y 143.522,Z 343.085,A -85,B 0,C 180,E1 -24598.917,E2 -24598.917} C_VEL
LIN {X 0,Y 146.189,Z 333.681,A -85,B 0,C 180,E1 -24601.52,E2 -24601.52} C_VEL
LIN {X 0,Y 148.752,Z 323.628,A -85,B 0,C 180,E1 -24603.72,E2 -24603.72} C_VEL
LIN {X 0,Y 151.367,Z 311.88,A -85,B 0,C 180,E1 -24605.681,E2 -24605.681} C_VEL
LIN {X 0,Y 153.705,Z 299.193,A -85,B 0,C 180,E1 -24607.186,E2 -24607.186} C_VEL
LIN {X 0,Y 155.324,Z 285.69,A -85,B 0,C 180,E1 -24608.266,E2 -24608.266} C_VEL
LIN {X 0,Y 157.413,Z 251.182,A -85,B 0,C 180,E1 -24609.8,E2 -24609.8} C_VEL
LIN {X 0,Y 157.78,Z 240.754,A -85,B 0,C 180,E1 -24610.288,E2 -24610.288} C_VEL
LIN {X 0,Y 156.024,Z 220.584,A -85,B 0,C 180,E1 -24611.832,E2 -24611.832} C_VEL
LIN {X 0,Y 150.94,Z 205.978,A -85,B 0,C 180,E1 -24613.99,E2 -24613.99} C_VEL
LIN {X 0,Y 144.847,Z 192.191,A -85,B 0,C 180,E1 -24616.617,E2 -24616.617} C_VEL
LIN {X 0,Y 141.196,Z 185.29,A -85,B 0,C 180,E1 -24618.258,E2 -24618.258} C_VEL
LIN {X 0,Y 138.817,Z 181.583,A -85,B 0,C 180,E1 -24619.341,E2 -24619.341} C_VEL
LIN {X 0,Y 136.571,Z 178.561,A -85,B 0,C 180,E1 -24620.382,E2 -24620.382} C_VEL
LIN {X 0,Y 136.007,Z 176.547,A -85,B 0,C 180,E1 -24620.814,E2 -24620.814} C_VEL
LIN {X 0,Y 136.057,Z 176.54,A -85,B 0,C 180,E1 -24625.737,E2 -24625.737} C_VEL
LIN {X 0,Y 136.146,Z 176.526,A -85,B 0,C 180,E1 -24632.316,E2 -24632.316} C_VEL
LIN {X 0,Y 136.234,Z 176.484,A -85,B 0,C 180,E1 -24638.831,E2 -24638.831} C_VEL
LIN {X 0,Y 136.233,Z 176.479,A -85,B 0,C 180,E1 -24645.051,E2 -24645.051} C_VEL
LIN {X 0,Y 136.425,Z 176.486,A -85,B 0,C 180,E1 -24648.177,E2 -24648.177} C_VEL
LIN {X 0,Y 136.547,Z 176.468,A -85,B 0,C 180,E1 -24651.117,E2 -24651.117} C_VEL
LIN {X 0,Y 137.132,Z 176.391,A -85,B 0,C 180,E1 -24659.999,E2 -24659.999} C_VEL
LIN {X 0,Y 136.551,Z 176.466,A -85,B 0,C 180,E1 -24668.882,E2 -24668.882} C_VEL
LIN {X 0,Y 136.44,Z 176.466,A -85,B 0,C 180,E1 -24671.89,E2 -24671.89} C_VEL
LIN {X 0,Y 136.241,Z 176.509,A -85,B 0,C 180,E1 -24678.029,E2 -24678.029} C_VEL
LIN {X 0,Y 136.195,Z 176.499,A -85,B 0,C 180,E1 -24681.746,E2 -24681.746} C_VEL
LIN {X 0,Y 136.097,Z 176.519,A -85,B 0,C 180,E1 -24688.614,E2 -24688.614} C_VEL
LIN {X 0,Y 136.041,Z 176.535,A -85,B 0,C 180,E1 -24694.629,E2 -24694.629} C_VEL
LIN {X 0,Y 136.03,Z 176.523,A -85,B 0,C 180,E1 -24699.198,E2 -24699.198} C_VEL
LIN {X 0,Y 135.996,Z 176.536,A -85,B 0,C 180,E1 -24703.657,E2 -24703.657} C_VEL
LIN {X 0,Y 136.027,Z 176.538,A -85,B 0,C 180,E1 -24707.805,E2 -24707.805} C_VEL
LIN {X 0,Y 136.025,Z 176.532,A -85,B 0,C 180,E1 -24711.684,E2 -24711.684} C_VEL
LIN {X 0,Y 136.054,Z 176.53,A -85,B 0,C 180,E1 -24715.739,E2 -24715.739} C_VEL
LIN {X 0,Y 136.084,Z 176.681,A -85,B 0,C 180,E1 -24720.049,E2 -24720.049} C_VEL
LIN {X 0,Y 137.099,Z 179.367,A -85,B 0,C 180,E1 -24720.627,E2 -24720.627} C_VEL
LIN {X 0,Y 139.043,Z 181.793,A -85,B 0,C 180,E1 -24721.508,E2 -24721.508} C_VEL
LIN {X 0,Y 147.541,Z 195.766,A -85,B 0,C 180,E1 -24725.182,E2 -24725.182} C_VEL
LIN {X 0,Y 153.478,Z 207.228,A -85,B 0,C 180,E1 -24727.515,E2 -24727.515} C_VEL
LIN {X 0,Y 158.962,Z 219.342,A -85,B 0,C 180,E1 -24729.558,E2 -24729.558} C_VEL
LIN {X 0,Y 155.815,Z 272.498,A -85,B 0,C 180,E1 -24731.838,E2 -24731.838} C_VEL
LIN {X 0,Y 154.38,Z 286.201,A -85,B 0,C 180,E1 -24732.94,E2 -24732.94} C_VEL
LIN {X 0,Y 152.476,Z 298.797,A -85,B 0,C 180,E1 -24734.46,E2 -24734.46} C_VEL
LIN {X 0,Y 150,Z 310.798,A -85,B 0,C 180,E1 -24736.452,E2 -24736.452} C_VEL
LIN {X 0,Y 147.168,Z 322.339,A -85,B 0,C 180,E1 -24738.988,E2 -24738.988} C_VEL
LIN {X 0,Y 144.29,Z 332.714,A -85,B 0,C 180,E1 -24741.951,E2 -24741.951} C_VEL
LIN {X 0,Y 141.205,Z 342.715,A -85,B 0,C 180,E1 -24745.643,E2 -24745.643} C_VEL
LIN {X 0,Y 138.872,Z 350.43,A -85,B 0,C 180,E1 -24749.276,E2 -24749.276} C_VEL
LIN {X 0,Y 136.646,Z 357.851,A -85,B 0,C 180,E1 -24753.687,E2 -24753.687} C_VEL
LIN {X 0,Y 134.966,Z 363.896,A -85,B 0,C 180,E1 -24758.363,E2 -24758.363} C_VEL
LIN {X 0,Y 133.802,Z 369.057,A -85,B 0,C 180,E1 -24763.673,E2 -24763.673} C_VEL
LIN {X 0,Y 133.313,Z 372.404,A -85,B 0,C 180,E1 -24768.44,E2 -24768.44} C_VEL
LIN {X 0,Y 133.383,Z 374.061,A -85,B 0,C 180,E1 -24771.644,E2 -24771.644} C_VEL
LIN {X 0,Y 134.181,Z 375.777,A -85,B 0,C 180,E1 -24777.076,E2 -24777.076} C_VEL
LIN {X 0,Y 135.413,Z 376.263,A -85,B 0,C 180,E1 -24781.266,E2 -24781.266} C_VEL
LIN {X 0,Y 136.973,Z 376.02,A -85,B 0,C 180,E1 -24784.821,E2 -24784.821} C_VEL
LIN {X 0,Y 140.51,Z 374.402,A -85,B 0,C 180,E1 -24790.56,E2 -24790.56} C_VEL
LIN {X 0,Y 144.17,Z 371.876,A -85,B 0,C 180,E1 -24794.98,E2 -24794.98} C_VEL
LIN {X 0,Y 148.654,Z 368.184,A -85,B 0,C 180,E1 -24799.152,E2 -24799.152} C_VEL
LIN {X 0,Y 153.554,Z 363.514,A -85,B 0,C 180,E1 -24802.871,E2 -24802.871} C_VEL
LIN {X 0,Y 159.702,Z 356.78,A -85,B 0,C 180,E1 -24806.735,E2 -24806.735} C_VEL
LIN {X 0,Y 165.933,Z 348.929,A -85,B 0,C 180,E1 -24810.015,E2 -24810.015} C_VEL
LIN {X 0,Y 171.98,Z 340.096,A -85,B 0,C 180,E1 -24812.726,E2 -24812.726} C_VEL
LIN {X 0,Y 177.451,Z 330.694,A -85,B 0,C 180,E1 -24814.951,E2 -24814.951} C_VEL
LIN {X 0,Y 182.539,Z 320.399,A -85,B 0,C 180,E1 -24816.813,E2 -24816.813} C_VEL
LIN {X 0,Y 187.182,Z 308.573,A -85,B 0,C 180,E1 -24818.469,E2 -24818.469} C_VEL
LIN {X 0,Y 191.052,Z 296.161,A -85,B 0,C 180,E1 -24819.726,E2 -24819.726} C_VEL
LIN {X 0,Y 193.892,Z 283.785,A -85,B 0,C 180,E1 -24820.618,E2 -24820.618} C_VEL
LIN {X 0,Y 195.715,Z 271.634,A -85,B 0,C 180,E1 -24821.196,E2 -24821.196} C_VEL
LIN {X 0,Y 197.371,Z 252.131,A -85,B 0,C 180,E1 -24821.863,E2 -24821.863} C_VEL
LIN {X 0,Y 193.037,Z 243.731,A -85,B 0,C 180,E1 -24824.958,E2 -24824.958} C_VEL
LIN {X 0,Y 189.577,Z 237.735,A -85,B 0,C 180,E1 -24827.747,E2 -24827.747} C_VEL
LIN {X 0,Y 186.161,Z 232.082,A -85,B 0,C 180,E1 -24830.963,E2 -24830.963} C_VEL
LIN {X 0,Y 183.484,Z 227.715,A -85,B 0,C 180,E1 -24834.065,E2 -24834.065} C_VEL
LIN {X 0,Y 181.227,Z 224.124,A -85,B 0,C 180,E1 -24837.291,E2 -24837.291} C_VEL
LIN {X 0,Y 179.264,Z 221.612,A -85,B 0,C 180,E1 -24840.948,E2 -24840.948} C_VEL
LIN {X 0,Y 178.459,Z 219.313,A -85,B 0,C 180,E1 -24843.535,E2 -24843.535} C_VEL
LIN {X 0,Y 177.394,Z 218.91,A -85,B 0,C 180,E1 -24849.119,E2 -24849.119} C_VEL
LIN {X 0,Y 178.215,Z 219.592,A -85,B 0,C 180,E1 -24855.262,E2 -24855.262} C_VEL
LIN {X 0,Y 179.324,Z 222.448,A -85,B 0,C 180,E1 -24858.814,E2 -24858.814} C_VEL
LIN {X 0,Y 180.316,Z 224.014,A -85,B 0,C 180,E1 -24860.804,E2 -24860.804} C_VEL
LIN {X 0,Y 181.657,Z 226.27,A -85,B 0,C 180,E1 -24863.039,E2 -24863.039} C_VEL
LIN {X 0,Y 184.552,Z 231.765,A -85,B 0,C 180,E1 -24866.963,E2 -24866.963} C_VEL
LIN {X 0,Y 187.135,Z 237.044,A -85,B 0,C 180,E1 -24869.793,E2 -24869.793} C_VEL
LIN {X 0,Y 190.437,Z 243.941,A -85,B 0,C 180,E1 -24872.836,E2 -24872.836} C_VEL
LIN {X 0,Y 193.914,Z 252.34,A -85,B 0,C 180,E1 -24875.695,E2 -24875.695} C_VEL
LIN {X 0,Y 196.751,Z 259.911,A -85,B 0,C 180,E1 -24877.812,E2 -24877.812} C_VEL
LIN {X 0,Y 194.578,Z 283.954,A -85,B 0,C 180,E1 -24878.648,E2 -24878.648} C_VEL
LIN {X 0,Y 191.949,Z 297.911,A -85,B 0,C 180,E1 -24879.331,E2 -24879.331} C_VEL
LIN {X 0,Y 188.651,Z 309.865,A -85,B 0,C 180,E1 -24880.207,E2 -24880.207} C_VEL
LIN {X 0,Y 184.148,Z 322.29,A -85,B 0,C 180,E1 -24881.497,E2 -24881.497} C_VEL
LIN {X 0,Y 179.134,Z 333.421,A -85,B 0,C 180,E1 -24883.053,E2 -24883.053} C_VEL
LIN {X 0,Y 173.671,Z 343.502,A -85,B 0,C 180,E1 -24884.912,E2 -24884.912} C_VEL
LIN {X 0,Y 168,Z 352.602,A -85,B 0,C 180,E1 -24887.172,E2 -24887.172} C_VEL
LIN {X 0,Y 161.579,Z 361.508,A -85,B 0,C 180,E1 -24890.091,E2 -24890.091} C_VEL
LIN {X 0,Y 155.634,Z 368.719,A -85,B 0,C 180,E1 -24893.249,E2 -24893.249} C_VEL
LIN {X 0,Y 151.131,Z 373.619,A -85,B 0,C 180,E1 -24896.079,E2 -24896.079} C_VEL
LIN {X 0,Y 146.742,Z 378.185,A -85,B 0,C 180,E1 -24899.553,E2 -24899.553} C_VEL
LIN {X 0,Y 142.47,Z 382.142,A -85,B 0,C 180,E1 -24903.642,E2 -24903.642} C_VEL
LIN {X 0,Y 140.115,Z 384.093,A -85,B 0,C 180,E1 -24906.342,E2 -24906.342} C_VEL
LIN {X 0,Y 138.12,Z 385.631,A -85,B 0,C 180,E1 -24909.133,E2 -24909.133} C_VEL
LIN {X 0,Y 136.436,Z 386.741,A -85,B 0,C 180,E1 -24911.996,E2 -24911.996} C_VEL
LIN {X 0,Y 134.396,Z 387.849,A -85,B 0,C 180,E1 -24917.926,E2 -24917.926} C_VEL
LIN {X 0,Y 133.738,Z 387.719,A -85,B 0,C 180,E1 -24921.842,E2 -24921.842} C_VEL
LIN {X 0,Y 133.718,Z 386.614,A -85,B 0,C 180,E1 -24926.987,E2 -24926.987} C_VEL
LIN {X 0,Y 133.905,Z 385.398,A -85,B 0,C 180,E1 -24929.999,E2 -24929.999} C_VEL
LIN {X 0,Y 133.682,Z 382.553,A -85,B 0,C 180,E1 -24934.705,E2 -24934.705} C_VEL
LIN {X 0,Y 133.065,Z 380.673,A -85,B 0,C 180,E1 -24937.091,E2 -24937.091} C_VEL
LIN {X 0,Y 130.594,Z 376.941,A -85,B 0,C 180,E1 -24940.952,E2 -24940.952} C_VEL
LIN {X 0,Y 128.555,Z 372.575,A -85,B 0,C 180,E1 -24944.812,E2 -24944.812} C_VEL
LIN {X 0,Y 128.632,Z 369.577,A -85,B 0,C 180,E1 -24947.097,E2 -24947.097} C_VEL
LIN {X 0,Y 130.57,Z 362.998,A -85,B 0,C 180,E1 -24951.304,E2 -24951.304} C_VEL
LIN {X 0,Y 133.089,Z 354.252,A -85,B 0,C 180,E1 -24955.692,E2 -24955.692} C_VEL
LIN {X 0,Y 136.383,Z 344.828,A -85,B 0,C 180,E1 -24959.31,E2 -24959.31} C_VEL
LIN {X 0,Y 139.096,Z 335.86,A -85,B 0,C 180,E1 -24962.04,E2 -24962.04} C_VEL
LIN {X 0,Y 141.226,Z 327.777,A -85,B 0,C 180,E1 -24964.045,E2 -24964.045} C_VEL
LIN {X 0,Y 144.142,Z 316.38,A -85,B 0,C 180,E1 -24966.24,E2 -24966.24} C_VEL
LIN {X 0,Y 146.577,Z 304.717,A -85,B 0,C 180,E1 -24967.902,E2 -24967.902} C_VEL
LIN {X 0,Y 148.581,Z 291.398,A -85,B 0,C 180,E1 -24969.232,E2 -24969.232} C_VEL
LIN {X 0,Y 149.837,Z 278.567,A -85,B 0,C 180,E1 -24970.025,E2 -24970.025} C_VEL
LIN {X 0,Y 151.841,Z 241.845,A -85,B 0,C 180,E1 -24971.656,E2 -24971.656} C_VEL
LIN {X 0,Y 150.275,Z 222.734,A -85,B 0,C 180,E1 -24973.173,E2 -24973.173} C_VEL
LIN {X 0,Y 145.409,Z 208.835,A -85,B 0,C 180,E1 -24975.384,E2 -24975.384} C_VEL
LIN {X 0,Y 140.114,Z 196.478,A -85,B 0,C 180,E1 -24977.864,E2 -24977.864} C_VEL
LIN {X 0,Y 136.686,Z 189.935,A -85,B 0,C 180,E1 -24979.522,E2 -24979.522} C_VEL
LIN {X 0,Y 133.297,Z 184.974,A -85,B 0,C 180,E1 -24981.172,E2 -24981.172} C_VEL
LIN {X 0,Y 131.397,Z 181.954,A -85,B 0,C 180,E1 -24982.162,E2 -24982.162} C_VEL
LIN {X 0,Y 129.554,Z 179.592,A -85,B 0,C 180,E1 -24983.121,E2 -24983.121} C_VEL
LIN {X 0,Y 128.933,Z 177.427,A -85,B 0,C 180,E1 -24983.643,E2 -24983.643} C_VEL
LIN {X 0,Y 128.979,Z 177.42,A -85,B 0,C 180,E1 -24986.982,E2 -24986.982} C_VEL
LIN {X 0,Y 129.051,Z 177.411,A -85,B 0,C 180,E1 -24990.65,E2 -24990.65} C_VEL
LIN {X 0,Y 129.105,Z 177.386,A -85,B 0,C 180,E1 -24997.729,E2 -24997.729} C_VEL
LIN {X 0,Y 129.157,Z 177.347,A -85,B 0,C 180,E1 -25004.212,E2 -25004.212} C_VEL
LIN {X 0,Y 129.345,Z 177.367,A -85,B 0,C 180,E1 -25007.967,E2 -25007.967} C_VEL
LIN {X 0,Y 129.47,Z 177.352,A -85,B 0,C 180,E1 -25010.627,E2 -25010.627} C_VEL
LIN {X 0,Y 130.087,Z 177.268,A -85,B 0,C 180,E1 -25019.999,E2 -25019.999} C_VEL
LIN {X 0,Y 129.474,Z 177.343,A -85,B 0,C 180,E1 -25029.371,E2 -25029.371} C_VEL
LIN {X 0,Y 129.344,Z 177.351,A -85,B 0,C 180,E1 -25032.552,E2 -25032.552} C_VEL
LIN {X 0,Y 129.151,Z 177.385,A -85,B 0,C 180,E1 -25039.056,E2 -25039.056} C_VEL
LIN {X 0,Y 129.107,Z 177.384,A -85,B 0,C 180,E1 -25042.398,E2 -25042.398} C_VEL
LIN {X 0,Y 129.026,Z 177.413,A -85,B 0,C 180,E1 -25045.833,E2 -25045.833} C_VEL
LIN {X 0,Y 129.015,Z 177.395,A -85,B 0,C 180,E1 -25049.358,E2 -25049.358} C_VEL
LIN {X 0,Y 128.958,Z 177.417,A -85,B 0,C 180,E1 -25055.168,E2 -25055.168} C_VEL
LIN {X 0,Y 128.942,Z 177.416,A -85,B 0,C 180,E1 -25060.848,E2 -25060.848} C_VEL
LIN {X 0,Y 128.92,Z 177.411,A -85,B 0,C 180,E1 -25065.127,E2 -25065.127} C_VEL
LIN {X 0,Y 128.946,Z 177.419,A -85,B 0,C 180,E1 -25069.733,E2 -25069.733} C_VEL
LIN {X 0,Y 128.958,Z 177.42,A -85,B 0,C 180,E1 -25074.832,E2 -25074.832} C_VEL
LIN {X 0,Y 128.986,Z 177.395,A -85,B 0,C 180,E1 -25077.164,E2 -25077.164} C_VEL
LIN {X 0,Y 129.924,Z 180.168,A -85,B 0,C 180,E1 -25077.828,E2 -25077.828} C_VEL
LIN {X 0,Y 132.066,Z 182.733,A -85,B 0,C 180,E1 -25078.919,E2 -25078.919} C_VEL
LIN {X 0,Y 134.395,Z 186.237,A -85,B 0,C 180,E1 -25080.099,E2 -25080.099} C_VEL
LIN {X 0,Y 141.518,Z 197.937,A -85,B 0,C 180,E1 -25083.452,E2 -25083.452} C_VEL
LIN {X 0,Y 147.11,Z 208.433,A -85,B 0,C 180,E1 -25085.842,E2 -25085.842} C_VEL
LIN {X 0,Y 152.972,Z 221.404,A -85,B 0,C 180,E1 -25088.206,E2 -25088.206} C_VEL
LIN {X 0,Y 149.783,Z 272.425,A -85,B 0,C 180,E1 -25090.436,E2 -25090.436} C_VEL
LIN {X 0,Y 148.334,Z 285.854,A -85,B 0,C 180,E1 -25091.53,E2 -25091.53} C_VEL
LIN {X 0,Y 146.514,Z 297.582,A -85,B 0,C 180,E1 -25092.947,E2 -25092.947} C_VEL
LIN {X 0,Y 144.161,Z 309.033,A -85,B 0,C 180,E1 -25094.81,E2 -25094.81} C_VEL
LIN {X 0,Y 141.149,Z 320.974,A -85,B 0,C 180,E1 -25097.418,E2 -25097.418} C_VEL
LIN {X 0,Y 138.089,Z 331.674,A -85,B 0,C 180,E1 -25100.48,E2 -25100.48} C_VEL
LIN {X 0,Y 135.029,Z 341.302,A -85,B 0,C 180,E1 -25104.025,E2 -25104.025} C_VEL
LIN {X 0,Y 132.038,Z 350.559,A -85,B 0,C 180,E1 -25108.476,E2 -25108.476} C_VEL
LIN {X 0,Y 129.682,Z 358.02,A -85,B 0,C 180,E1 -25113.107,E2 -25113.107} C_VEL
LIN {X 0,Y 127.832,Z 364.35,A -85,B 0,C 180,E1 -25118.269,E2 -25118.269} C_VEL
LIN {X 0,Y 126.832,Z 368.629,A -85,B 0,C 180,E1 -25122.806,E2 -25122.806} C_VEL
LIN {X 0,Y 126.397,Z 371.109,A -85,B 0,C 180,E1 -25126.142,E2 -25126.142} C_VEL
LIN {X 0,Y 126.193,Z 373.144,A -85,B 0,C 180,E1 -25129.522,E2 -25129.522} C_VEL
LIN {X 0,Y 126.4,Z 374.658,A -85,B 0,C 180,E1 -25132.906,E2 -25132.906} C_VEL
LIN {X 0,Y 127.285,Z 376.112,A -85,B 0,C 180,E1 -25137.941,E2 -25137.941} C_VEL
LIN {X 0,Y 128.916,Z 376.581,A -85,B 0,C 180,E1 -25143.036,E2 -25143.036} C_VEL
LIN {X 0,Y 130.503,Z 376.316,A -85,B 0,C 180,E1 -25146.327,E2 -25146.327} C_VEL
LIN {X 0,Y 132.437,Z 375.624,A -85,B 0,C 180,E1 -25149.554,E2 -25149.554} C_VEL
LIN {X 0,Y 135.19,Z 374.137,A -85,B 0,C 180,E1 -25153.298,E2 -25153.298} C_VEL
LIN {X 0,Y 140.35,Z 370.61,A -85,B 0,C 180,E1 -25158.688,E2 -25158.688} C_VEL
LIN {X 0,Y 145.522,Z 366.324,A -85,B 0,C 180,E1 -25162.833,E2 -25162.833} C_VEL
LIN {X 0,Y 151.389,Z 360.683,A -85,B 0,C 180,E1 -25166.682,E2 -25166.682} C_VEL
LIN {X 0,Y 157.601,Z 353.756,A -85,B 0,C 180,E1 -25170.141,E2 -25170.141} C_VEL
LIN {X 0,Y 163.667,Z 346.017,A -85,B 0,C 180,E1 -25173.003,E2 -25173.003} C_VEL
LIN {X 0,Y 169.985,Z 336.619,A -85,B 0,C 180,E1 -25175.579,E2 -25175.579} C_VEL
LIN {X 0,Y 175.661,Z 326.536,A -85,B 0,C 180,E1 -25177.7,E2 -25177.7} C_VEL
LIN {X 0,Y 181.049,Z 314.926,A -85,B 0,C 180,E1 -25179.552,E2 -25179.552} C_VEL
LIN {X 0,Y 185.409,Z 303.05,A -85,B 0,C 180,E1 -25180.956,E2 -25180.956} C_VEL
LIN {X 0,Y 188.899,Z 290.561,A -85,B 0,C 180,E1 -25182.047,E2 -25182.047} C_VEL
LIN {X 0,Y 191.461,Z 277.441,A -85,B 0,C 180,E1 -25182.805,E2 -25182.805} C_VEL
LIN {X 0,Y 193.449,Z 259.217,A -85,B 0,C 180,E1 -25183.424,E2 -25183.424} C_VEL
LIN {X 0,Y 193.703,Z 255.71,A -85,B 0,C 180,E1 -25183.566,E2 -25183.566} C_VEL
LIN {X 0,Y 189.771,Z 247.898,A -85,B 0,C 180,E1 -25186.648,E2 -25186.648} C_VEL
LIN {X 0,Y 185.89,Z 241.081,A -85,B 0,C 180,E1 -25190.159,E2 -25190.159} C_VEL
LIN {X 0,Y 183.937,Z 237.84,A -85,B 0,C 180,E1 -25192.264,E2 -25192.264} C_VEL
LIN {X 0,Y 181.931,Z 234.255,A -85,B 0,C 180,E1 -25194.804,E2 -25194.804} C_VEL
LIN {X 0,Y 179.839,Z 230.859,A -85,B 0,C 180,E1 -25197.986,E2 -25197.986} C_VEL
LIN {X 0,Y 177.982,Z 228.08,A -85,B 0,C 180,E1 -25201.892,E2 -25201.892} C_VEL
LIN {X 0,Y 177.53,Z 226.475,A -85,B 0,C 180,E1 -25203.553,E2 -25203.553} C_VEL
LIN {X 0,Y 176.491,Z 225.948,A -85,B 0,C 180,E1 -25209.166,E2 -25209.166} C_VEL
LIN {X 0,Y 177.207,Z 226.594,A -85,B 0,C 180,E1 -25214.913,E2 -25214.913} C_VEL
LIN {X 0,Y 178.381,Z 229.536,A -85,B 0,C 180,E1 -25218.767,E2 -25218.767} C_VEL
LIN {X 0,Y 180.243,Z 232.904,A -85,B 0,C 180,E1 -25222.345,E2 -25222.345} C_VEL
LIN {X 0,Y 182.867,Z 238.148,A -85,B 0,C 180,E1 -25226.154,E2 -25226.154} C_VEL
LIN {X 0,Y 185.182,Z 243.272,A -85,B 0,C 180,E1 -25228.915,E2 -25228.915} C_VEL
LIN {X 0,Y 188.081,Z 249.657,A -85,B 0,C 180,E1 -25231.779,E2 -25231.779} C_VEL
LIN {X 0,Y 191.175,Z 257.576,A -85,B 0,C 180,E1 -25234.524,E2 -25234.524} C_VEL
LIN {X 0,Y 193.077,Z 262.874,A -85,B 0,C 180,E1 -25236.082,E2 -25236.082} C_VEL
LIN {X 0,Y 191.241,Z 282.426,A -85,B 0,C 180,E1 -25236.745,E2 -25236.745} C_VEL
LIN {X 0,Y 188.73,Z 296.055,A -85,B 0,C 180,E1 -25237.395,E2 -25237.395} C_VEL
LIN {X 0,Y 185.218,Z 308.815,A -85,B 0,C 180,E1 -25238.281,E2 -25238.281} C_VEL
LIN {X 0,Y 180.888,Z 320.609,A -85,B 0,C 180,E1 -25239.448,E2 -25239.448} C_VEL
LIN {X 0,Y 175.681,Z 331.979,A -85,B 0,C 180,E1 -25240.967,E2 -25240.967} C_VEL
LIN {X 0,Y 170.014,Z 342.277,A -85,B 0,C 180,E1 -25242.798,E2 -25242.798} C_VEL
LIN {X 0,Y 164.075,Z 351.568,A -85,B 0,C 180,E1 -25245.027,E2 -25245.027} C_VEL
LIN {X 0,Y 157.338,Z 360.591,A -85,B 0,C 180,E1 -25247.931,E2 -25247.931} C_VEL
LIN {X 0,Y 151.015,Z 367.906,A -85,B 0,C 180,E1 -25251.077,E2 -25251.077} C_VEL
LIN {X 0,Y 145.298,Z 373.805,A -85,B 0,C 180,E1 -25254.518,E2 -25254.518} C_VEL
LIN {X 0,Y 140.347,Z 378.559,A -85,B 0,C 180,E1 -25258.353,E2 -25258.353} C_VEL
LIN {X 0,Y 136.141,Z 382.117,A -85,B 0,C 180,E1 -25262.315,E2 -25262.315} C_VEL
LIN {X 0,Y 133.614,Z 384.014,A -85,B 0,C 180,E1 -25265.115,E2 -25265.115} C_VEL
LIN {X 0,Y 129.673,Z 386.527,A -85,B 0,C 180,E1 -25271.023,E2 -25271.023} C_VEL
LIN {X 0,Y 127.427,Z 387.545,A -85,B 0,C 180,E1 -25277.254,E2 -25277.254} C_VEL
LIN {X 0,Y 126.83,Z 387.47,A -85,B 0,C 180,E1 -25280.43,E2 -25280.43} C_VEL
LIN {X 0,Y 126.637,Z 386.139,A -85,B 0,C 180,E1 -25286.818,E2 -25286.818} C_VEL
LIN {X 0,Y 126.809,Z 384.881,A -85,B 0,C 180,E1 -25289.999,E2 -25289.999} C_VEL
LIN {X 0,Y 126.613,Z 382.083,A -85,B 0,C 180,E1 -25294.775,E2 -25294.775} C_VEL
LIN {X 0,Y 126.872,Z 378.209,A -85,B 0,C 180,E1 -25299.565,E2 -25299.565} C_VEL
LIN {X 0,Y 127.762,Z 373.16,A -85,B 0,C 180,E1 -25304.331,E2 -25304.331} C_VEL
LIN {X 0,Y 128.632,Z 369.577,A -85,B 0,C 180,E1 -25307.097,E2 -25307.097} C_VEL
LIN {X 0,Y 128.839,Z 366.39,A -85,B 0,C 180,E1 -25309.306,E2 -25309.306} C_VEL
LIN {X 0,Y 127.667,Z 360.669,A -85,B 0,C 180,E1 -25312.911,E2 -25312.911} C_VEL
LIN {X 0,Y 126.921,Z 354.407,A -85,B 0,C 180,E1 -25316.364,E2 -25316.364} C_VEL
LIN {X 0,Y 127.761,Z 350.286,A -85,B 0,C 180,E1 -25318.234,E2 -25318.234} C_VEL
LIN {X 0,Y 130.778,Z 341.141,A -85,B 0,C 180,E1 -25321.598,E2 -25321.598} C_VEL
LIN {X 0,Y 133.37,Z 332.776,A -85,B 0,C 180,E1 -25324.047,E2 -25324.047} C_VEL
LIN {X 0,Y 136.666,Z 321.083,A -85,B 0,C 180,E1 -25326.713,E2 -25326.713} C_VEL
LIN {X 0,Y 139.555,Z 308.667,A -85,B 0,C 180,E1 -25328.781,E2 -25328.781} C_VEL
LIN {X 0,Y 141.861,Z 295.893,A -85,B 0,C 180,E1 -25330.284,E2 -25330.284} C_VEL
LIN {X 0,Y 143.465,Z 283.223,A -85,B 0,C 180,E1 -25331.261,E2 -25331.261} C_VEL
LIN {X 0,Y 145.938,Z 242.649,A -85,B 0,C 180,E1 -25333.139,E2 -25333.139} C_VEL
LIN {X 0,Y 144.493,Z 224.708,A -85,B 0,C 180,E1 -25334.655,E2 -25334.655} C_VEL
LIN {X 0,Y 140.18,Z 212.137,A -85,B 0,C 180,E1 -25336.79,E2 -25336.79} C_VEL
LIN {X 0,Y 135.312,Z 200.486,A -85,B 0,C 180,E1 -25339.27,E2 -25339.27} C_VEL
LIN {X 0,Y 132.314,Z 194.652,A -85,B 0,C 180,E1 -25340.84,E2 -25340.84} C_VEL
LIN {X 0,Y 127.248,Z 186.994,A -85,B 0,C 180,E1 -25343.547,E2 -25343.547} C_VEL
LIN {X 0,Y 125.146,Z 183.762,A -85,B 0,C 180,E1 -25344.779,E2 -25344.779} C_VEL
LIN {X 0,Y 124.145,Z 182.65,A -85,B 0,C 180,E1 -25345.352,E2 -25345.352} C_VEL
LIN {X 0,Y 122.509,Z 180.396,A -85,B 0,C 180,E1 -25346.361,E2 -25346.361} C_VEL
LIN {X 0,Y 121.931,Z 178.297,A -85,B 0,C 180,E1 -25346.922,E2 -25346.922} C_VEL
LIN {X 0,Y 121.956,Z 178.294,A -85,B 0,C 180,E1 -25352.546,E2 -25352.546} C_VEL
LIN {X 0,Y 122.022,Z 178.274,A -85,B 0,C 180,E1 -25357.151,E2 -25357.151} C_VEL
LIN {X 0,Y 122.074,Z 178.22,A -85,B 0,C 180,E1 -25363.27,E2 -25363.27} C_VEL
LIN {X 0,Y 122.287,Z 178.243,A -85,B 0,C 180,E1 -25367.687,E2 -25367.687} C_VEL
LIN {X 0,Y 122.396,Z 178.236,A -85,B 0,C 180,E1 -25370.08,E2 -25370.08} C_VEL
LIN {X 0,Y 122.593,Z 178.207,A -85,B 0,C 180,E1 -25376.713,E2 -25376.713} C_VEL
LIN {X 0,Y 123.04,Z 178.145,A -85,B 0,C 180,E1 -25379.999,E2 -25379.999} C_VEL
LIN {X 0,Y 122.405,Z 178.23,A -85,B 0,C 180,E1 -25386.917,E2 -25386.917} C_VEL
LIN {X 0,Y 122.322,Z 178.224,A -85,B 0,C 180,E1 -25392.386,E2 -25392.386} C_VEL
LIN {X 0,Y 122.107,Z 178.274,A -85,B 0,C 180,E1 -25396.724,E2 -25396.724} C_VEL
LIN {X 0,Y 122.026,Z 178.268,A -85,B 0,C 180,E1 -25402.854,E2 -25402.854} C_VEL
LIN {X 0,Y 121.939,Z 178.289,A -85,B 0,C 180,E1 -25407.456,E2 -25407.456} C_VEL
LIN {X 0,Y 121.898,Z 178.28,A -85,B 0,C 180,E1 -25411.257,E2 -25411.257} C_VEL
LIN {X 0,Y 121.882,Z 178.293,A -85,B 0,C 180,E1 -25416.171,E2 -25416.171} C_VEL
LIN {X 0,Y 121.878,Z 178.298,A -85,B 0,C 180,E1 -25421.442,E2 -25421.442} C_VEL
LIN {X 0,Y 121.878,Z 178.302,A -85,B 0,C 180,E1 -25428.558,E2 -25428.558} C_VEL
LIN {X 0,Y 121.901,Z 178.38,A -85,B 0,C 180,E1 -25433.904,E2 -25433.904} C_VEL
LIN {X 0,Y 122.768,Z 180.867,A -85,B 0,C 180,E1 -25434.571,E2 -25434.571} C_VEL
LIN {X 0,Y 124.757,Z 183.115,A -85,B 0,C 180,E1 -25435.741,E2 -25435.741} C_VEL
LIN {X 0,Y 127.36,Z 187.086,A -85,B 0,C 180,E1 -25437.267,E2 -25437.267} C_VEL
LIN {X 0,Y 132.642,Z 195.063,A -85,B 0,C 180,E1 -25440.069,E2 -25440.069} C_VEL
LIN {X 0,Y 139.482,Z 207.071,A -85,B 0,C 180,E1 -25443.392,E2 -25443.392} C_VEL
LIN {X 0,Y 145.453,Z 219.795,A -85,B 0,C 180,E1 -25446.069,E2 -25446.069} C_VEL
LIN {X 0,Y 147.076,Z 223.808,A -85,B 0,C 180,E1 -25446.778,E2 -25446.778} C_VEL
LIN {X 0,Y 143.704,Z 273.579,A -85,B 0,C 180,E1 -25449.012,E2 -25449.012} C_VEL
LIN {X 0,Y 142.096,Z 287.438,A -85,B 0,C 180,E1 -25450.212,E2 -25450.212} C_VEL
LIN {X 0,Y 139.94,Z 300.108,A -85,B 0,C 180,E1 -25451.869,E2 -25451.869} C_VEL
LIN {X 0,Y 137.228,Z 312.075,A -85,B 0,C 180,E1 -25454.022,E2 -25454.022} C_VEL
LIN {X 0,Y 134.121,Z 323.505,A -85,B 0,C 180,E1 -25456.748,E2 -25456.748} C_VEL
LIN {X 0,Y 130.98,Z 333.75,A -85,B 0,C 180,E1 -25459.958,E2 -25459.958} C_VEL
LIN {X 0,Y 127.812,Z 343.031,A -85,B 0,C 180,E1 -25463.687,E2 -25463.687} C_VEL
LIN {X 0,Y 124.76,Z 352.055,A -85,B 0,C 180,E1 -25468.387,E2 -25468.387} C_VEL
LIN {X 0,Y 122.398,Z 359.239,A -85,B 0,C 180,E1 -25473.292,E2 -25473.292} C_VEL
LIN {X 0,Y 120.707,Z 364.819,A -85,B 0,C 180,E1 -25478.194,E2 -25478.194} C_VEL
LIN {X 0,Y 119.586,Z 369.515,A -85,B 0,C 180,E1 -25483.597,E2 -25483.597} C_VEL
LIN {X 0,Y 119.116,Z 373.094,A -85,B 0,C 180,E1 -25489.264,E2 -25489.264} C_VEL
LIN {X 0,Y 119.44,Z 375.255,A -85,B 0,C 180,E1 -25494.324,E2 -25494.324} C_VEL
LIN {X 0,Y 120.382,Z 376.443,A -85,B 0,C 180,E1 -25498.872,E2 -25498.872} C_VEL
LIN {X 0,Y 122.557,Z 376.891,A -85,B 0,C 180,E1 -25504.992,E2 -25504.992} C_VEL
LIN {X 0,Y 124.38,Z 376.555,A -85,B 0,C 180,E1 -25508.43,E2 -25508.43} C_VEL
LIN {X 0,Y 126.566,Z 375.731,A -85,B 0,C 180,E1 -25511.786,E2 -25511.786} C_VEL
LIN {X 0,Y 129.138,Z 374.44,A -85,B 0,C 180,E1 -25515.032,E2 -25515.032} C_VEL
LIN {X 0,Y 133.684,Z 371.598,A -85,B 0,C 180,E1 -25519.667,E2 -25519.667} C_VEL
LIN {X 0,Y 139.043,Z 367.573,A -85,B 0,C 180,E1 -25523.972,E2 -25523.972} C_VEL
LIN {X 0,Y 145.796,Z 361.579,A -85,B 0,C 180,E1 -25528.33,E2 -25528.33} C_VEL
LIN {X 0,Y 151.805,Z 355.332,A -85,B 0,C 180,E1 -25531.598,E2 -25531.598} C_VEL
LIN {X 0,Y 157.821,Z 348.204,A -85,B 0,C 180,E1 -25534.391,E2 -25534.391} C_VEL
LIN {X 0,Y 163.941,Z 339.914,A -85,B 0,C 180,E1 -25536.833,E2 -25536.833} C_VEL
LIN {X 0,Y 170.188,Z 329.852,A -85,B 0,C 180,E1 -25539.118,E2 -25539.118} C_VEL
LIN {X 0,Y 175.639,Z 319.22,A -85,B 0,C 180,E1 -25540.921,E2 -25540.921} C_VEL
LIN {X 0,Y 179.856,Z 309.126,A -85,B 0,C 180,E1 -25542.266,E2 -25542.266} C_VEL
LIN {X 0,Y 183.82,Z 297.263,A -85,B 0,C 180,E1 -25543.447,E2 -25543.447} C_VEL
LIN {X 0,Y 186.958,Z 284.601,A -85,B 0,C 180,E1 -25544.343,E2 -25544.343} C_VEL
LIN {X 0,Y 188.832,Z 273.222,A -85,B 0,C 180,E1 -25544.884,E2 -25544.884} C_VEL
LIN {X 0,Y 190.165,Z 259.246,A -85,B 0,C 180,E1 -25545.366,E2 -25545.366} C_VEL
LIN {X 0,Y 186.347,Z 251.555,A -85,B 0,C 180,E1 -25548.692,E2 -25548.692} C_VEL
LIN {X 0,Y 182.906,Z 245.225,A -85,B 0,C 180,E1 -25552.298,E2 -25552.298} C_VEL
LIN {X 0,Y 180.337,Z 240.737,A -85,B 0,C 180,E1 -25555.648,E2 -25555.648} C_VEL
LIN {X 0,Y 178.637,Z 237.735,A -85,B 0,C 180,E1 -25558.426,E2 -25558.426} C_VEL
LIN {X 0,Y 176.823,Z 234.734,A -85,B 0,C 180,E1 -25562.601,E2 -25562.601} C_VEL
LIN {X 0,Y 176.461,Z 233.426,A -85,B 0,C 180,E1 -25564.072,E2 -25564.072} C_VEL
LIN {X 0,Y 175.587,Z 232.993,A -85,B 0,C 180,E1 -25569.213,E2 -25569.213} C_VEL
LIN {X 0,Y 176.195,Z 233.565,A -85,B 0,C 180,E1 -25574.506,E2 -25574.506} C_VEL
LIN {X 0,Y 178.057,Z 237.952,A -85,B 0,C 180,E1 -25580.121,E2 -25580.121} C_VEL
LIN {X 0,Y 178.988,Z 239.861,A -85,B 0,C 180,E1 -25581.884,E2 -25581.884} C_VEL
LIN {X 0,Y 181.215,Z 244.573,A -85,B 0,C 180,E1 -25585.33,E2 -25585.33} C_VEL
LIN {X 0,Y 183.169,Z 249.183,A -85,B 0,C 180,E1 -25587.862,E2 -25587.862} C_VEL
LIN {X 0,Y 185.929,Z 255.783,A -85,B 0,C 180,E1 -25590.841,E2 -25590.841} C_VEL
LIN {X 0,Y 189.043,Z 264.236,A -85,B 0,C 180,E1 -25593.788,E2 -25593.788} C_VEL
LIN {X 0,Y 189.624,Z 266.043,A -85,B 0,C 180,E1 -25594.313,E2 -25594.313} C_VEL
LIN {X 0,Y 187.62,Z 284.691,A -85,B 0,C 180,E1 -25594.953,E2 -25594.953} C_VEL
LIN {X 0,Y 184.972,Z 297.525,A -85,B 0,C 180,E1 -25595.558,E2 -25595.558} C_VEL
LIN {X 0,Y 181.287,Z 309.917,A -85,B 0,C 180,E1 -25596.445,E2 -25596.445} C_VEL
LIN {X 0,Y 176.516,Z 322.173,A -85,B 0,C 180,E1 -25597.69,E2 -25597.69} C_VEL
LIN {X 0,Y 171.151,Z 333.192,A -85,B 0,C 180,E1 -25599.188,E2 -25599.188} C_VEL
LIN {X 0,Y 165.309,Z 343.149,A -85,B 0,C 180,E1 -25601.006,E2 -25601.006} C_VEL
LIN {X 0,Y 159.158,Z 352.184,A -85,B 0,C 180,E1 -25603.23,E2 -25603.23} C_VEL
LIN {X 0,Y 152.159,Z 361.033,A -85,B 0,C 180,E1 -25606.145,E2 -25606.145} C_VEL
LIN {X 0,Y 145.571,Z 368.21,A -85,B 0,C 180,E1 -25609.325,E2 -25609.325} C_VEL
LIN {X 0,Y 139.575,Z 373.98,A -85,B 0,C 180,E1 -25612.826,E2 -25612.826} C_VEL
LIN {X 0,Y 133.868,Z 378.985,A -85,B 0,C 180,E1 -25617.14,E2 -25617.14} C_VEL
LIN {X 0,Y 129.891,Z 382.093,A -85,B 0,C 180,E1 -25620.858,E2 -25620.858} C_VEL
LIN {X 0,Y 127.183,Z 383.9,A -85,B 0,C 180,E1 -25623.763,E2 -25623.763} C_VEL
LIN {X 0,Y 122.959,Z 386.315,A -85,B 0,C 180,E1 -25629.943,E2 -25629.943} C_VEL
LIN {X 0,Y 120.487,Z 387.223,A -85,B 0,C 180,E1 -25636.507,E2 -25636.507} C_VEL
LIN {X 0,Y 119.502,Z 386.553,A -85,B 0,C 180,E1 -25643.245,E2 -25643.245} C_VEL
LIN {X 0,Y 119.586,Z 385.35,A -85,B 0,C 180,E1 -25647.555,E2 -25647.555} C_VEL
LIN {X 0,Y 119.734,Z 384.348,A -85,B 0,C 180,E1 -25649.999,E2 -25649.999} C_VEL
LIN {X 0,Y 119.531,Z 381.456,A -85,B 0,C 180,E1 -25655.059,E2 -25655.059} C_VEL
LIN {X 0,Y 119.842,Z 377.479,A -85,B 0,C 180,E1 -25660.132,E2 -25660.132} C_VEL
LIN {X 0,Y 121.09,Z 371.298,A -85,B 0,C 180,E1 -25666.002,E2 -25666.002} C_VEL
LIN {X 0,Y 123.127,Z 364.523,A -85,B 0,C 180,E1 -25670.9,E2 -25670.9} C_VEL
LIN {X 0,Y 125.759,Z 356.046,A -85,B 0,C 180,E1 -25675.664,E2 -25675.664} C_VEL
LIN {X 0,Y 127.761,Z 350.286,A -85,B 0,C 180,E1 -25678.234,E2 -25678.234} C_VEL
LIN {X 0,Y 128.642,Z 346.018,A -85,B 0,C 180,E1 -25680,E2 -25680} C_VEL
LIN {X 0,Y 128.311,Z 338.682,A -85,B 0,C 180,E1 -25682.977,E2 -25682.977} C_VEL
LIN {X 0,Y 128.076,Z 330.9,A -85,B 0,C 180,E1 -25685.747,E2 -25685.747} C_VEL
LIN {X 0,Y 129.058,Z 325.849,A -85,B 0,C 180,E1 -25687.105,E2 -25687.105} C_VEL
LIN {X 0,Y 131.931,Z 315.239,A -85,B 0,C 180,E1 -25689.24,E2 -25689.24} C_VEL
LIN {X 0,Y 134.596,Z 303.361,A -85,B 0,C 180,E1 -25690.992,E2 -25690.992} C_VEL
LIN {X 0,Y 136.788,Z 289.781,A -85,B 0,C 180,E1 -25692.385,E2 -25692.385} C_VEL
LIN {X 0,Y 138.04,Z 277.115,A -85,B 0,C 180,E1 -25693.187,E2 -25693.187} C_VEL
LIN {X 0,Y 140.093,Z 243.146,A -85,B 0,C 180,E1 -25694.779,E2 -25694.779} C_VEL
LIN {X 0,Y 138.957,Z 227.054,A -85,B 0,C 180,E1 -25696.189,E2 -25696.189} C_VEL
LIN {X 0,Y 134.908,Z 215.074,A -85,B 0,C 180,E1 -25698.377,E2 -25698.377} C_VEL
LIN {X 0,Y 130.65,Z 204.604,A -85,B 0,C 180,E1 -25700.749,E2 -25700.749} C_VEL
LIN {X 0,Y 127.953,Z 199.291,A -85,B 0,C 180,E1 -25702.264,E2 -25702.264} C_VEL
LIN {X 0,Y 123.353,Z 192.177,A -85,B 0,C 180,E1 -25704.916,E2 -25704.916} C_VEL
LIN {X 0,Y 120.745,Z 188.355,A -85,B 0,C 180,E1 -25706.554,E2 -25706.554} C_VEL
LIN {X 0,Y 118.509,Z 185.04,A -85,B 0,C 180,E1 -25708.064,E2 -25708.064} C_VEL
LIN {X 0,Y 117.952,Z 184.198,A -85,B 0,C 180,E1 -25708.457,E2 -25708.457} C_VEL
LIN {X 0,Y 115.866,Z 181.979,A -85,B 0,C 180,E1 -25709.901,E2 -25709.901} C_VEL
LIN {X 0,Y 114.87,Z 179.176,A -85,B 0,C 180,E1 -25710.82,E2 -25710.82} C_VEL
LIN {X 0,Y 114.945,Z 179.161,A -85,B 0,C 180,E1 -25716.509,E2 -25716.509} C_VEL
LIN {X 0,Y 114.982,Z 179.098,A -85,B 0,C 180,E1 -25722.204,E2 -25722.204} C_VEL
LIN {X 0,Y 115.309,Z 179.119,A -85,B 0,C 180,E1 -25729.464,E2 -25729.464} C_VEL
LIN {X 0,Y 115.517,Z 179.087,A -85,B 0,C 180,E1 -25736.511,E2 -25736.511} C_VEL
LIN {X 0,Y 115.992,Z 179.022,A -85,B 0,C 180,E1 -25739.999,E2 -25739.999} C_VEL
LIN {X 0,Y 115.365,Z 179.11,A -85,B 0,C 180,E1 -25746.998,E2 -25746.998} C_VEL
LIN {X 0,Y 115.254,Z 179.105,A -85,B 0,C 180,E1 -25752.673,E2 -25752.673} C_VEL
LIN {X 0,Y 115.01,Z 179.154,A -85,B 0,C 180,E1 -25757.79,E2 -25757.79} C_VEL
LIN {X 0,Y 114.946,Z 179.155,A -85,B 0,C 180,E1 -25763.492,E2 -25763.492} C_VEL
LIN {X 0,Y 114.855,Z 179.156,A -85,B 0,C 180,E1 -25771.057,E2 -25771.057} C_VEL
LIN {X 0,Y 114.779,Z 179.167,A -85,B 0,C 180,E1 -25777.756,E2 -25777.756} C_VEL
LIN {X 0,Y 114.79,Z 179.182,A -85,B 0,C 180,E1 -25782.719,E2 -25782.719} C_VEL
LIN {X 0,Y 114.829,Z 179.176,A -85,B 0,C 180,E1 -25789.844,E2 -25789.844} C_VEL
LIN {X 0,Y 115.898,Z 182.172,A -85,B 0,C 180,E1 -25790.889,E2 -25790.889} C_VEL
LIN {X 0,Y 118.161,Z 184.38,A -85,B 0,C 180,E1 -25792.434,E2 -25792.434} C_VEL
LIN {X 0,Y 120.476,Z 188.06,A -85,B 0,C 180,E1 -25794.037,E2 -25794.037} C_VEL
LIN {X 0,Y 121.667,Z 189.59,A -85,B 0,C 180,E1 -25794.788,E2 -25794.788} C_VEL
LIN {X 0,Y 127.304,Z 198.089,A -85,B 0,C 180,E1 -25798.127,E2 -25798.127} C_VEL
LIN {X 0,Y 134.075,Z 210.005,A -85,B 0,C 180,E1 -25801.708,E2 -25801.708} C_VEL
LIN {X 0,Y 138.927,Z 220.213,A -85,B 0,C 180,E1 -25804.094,E2 -25804.094} C_VEL
LIN {X 0,Y 141.114,Z 225.308,A -85,B 0,C 180,E1 -25805.124,E2 -25805.124} C_VEL
LIN {X 0,Y 137.86,Z 273.506,A -85,B 0,C 180,E1 -25807.379,E2 -25807.379} C_VEL
LIN {X 0,Y 136.255,Z 287.011,A -85,B 0,C 180,E1 -25808.565,E2 -25808.565} C_VEL
LIN {X 0,Y 134.136,Z 299.169,A -85,B 0,C 180,E1 -25810.149,E2 -25810.149} C_VEL
LIN {X 0,Y 131.563,Z 310.276,A -85,B 0,C 180,E1 -25812.112,E2 -25812.112} C_VEL
LIN {X 0,Y 128.249,Z 322.093,A -85,B 0,C 180,E1 -25814.913,E2 -25814.913} C_VEL
LIN {X 0,Y 124.896,Z 332.709,A -85,B 0,C 180,E1 -25818.231,E2 -25818.231} C_VEL
LIN {X 0,Y 121.851,Z 341.392,A -85,B 0,C 180,E1 -25821.71,E2 -25821.71} C_VEL
LIN {X 0,Y 118.907,Z 349.429,A -85,B 0,C 180,E1 -25825.799,E2 -25825.799} C_VEL
LIN {X 0,Y 116.213,Z 357.14,A -85,B 0,C 180,E1 -25830.867,E2 -25830.867} C_VEL
LIN {X 0,Y 114.44,Z 362.456,A -85,B 0,C 180,E1 -25835.286,E2 -25835.286} C_VEL
LIN {X 0,Y 112.988,Z 367.606,A -85,B 0,C 180,E1 -25840.755,E2 -25840.755} C_VEL
LIN {X 0,Y 112.157,Z 371.593,A -85,B 0,C 180,E1 -25846.379,E2 -25846.379} C_VEL
LIN {X 0,Y 112.09,Z 374.488,A -85,B 0,C 180,E1 -25852.099,E2 -25852.099} C_VEL
LIN {X 0,Y 112.572,Z 375.853,A -85,B 0,C 180,E1 -25855.915,E2 -25855.915} C_VEL
LIN {X 0,Y 113.499,Z 376.772,A -85,B 0,C 180,E1 -25859.901,E2 -25859.901} C_VEL
LIN {X 0,Y 114.677,Z 377.185,A -85,B 0,C 180,E1 -25863.475,E2 -25863.475} C_VEL
LIN {X 0,Y 117.256,Z 377.037,A -85,B 0,C 180,E1 -25868.815,E2 -25868.815} C_VEL
LIN {X 0,Y 120.91,Z 375.822,A -85,B 0,C 180,E1 -25874.229,E2 -25874.229} C_VEL
LIN {X 0,Y 123.796,Z 374.456,A -85,B 0,C 180,E1 -25877.564,E2 -25877.564} C_VEL
LIN {X 0,Y 128.787,Z 371.486,A -85,B 0,C 180,E1 -25882.252,E2 -25882.252} C_VEL
LIN {X 0,Y 134.664,Z 367.263,A -85,B 0,C 180,E1 -25886.62,E2 -25886.62} C_VEL
LIN {X 0,Y 141.427,Z 361.49,A -85,B 0,C 180,E1 -25890.711,E2 -25890.711} C_VEL
LIN {X 0,Y 148.31,Z 354.607,A -85,B 0,C 180,E1 -25894.206,E2 -25894.206} C_VEL
LIN {X 0,Y 154.677,Z 347.263,A -85,B 0,C 180,E1 -25896.941,E2 -25896.941} C_VEL
LIN {X 0,Y 161.437,Z 338.174,A -85,B 0,C 180,E1 -25899.461,E2 -25899.461} C_VEL
LIN {X 0,Y 167.615,Z 328.172,A -85,B 0,C 180,E1 -25901.561,E2 -25901.561} C_VEL
LIN {X 0,Y 173.296,Z 317.025,A -85,B 0,C 180,E1 -25903.34,E2 -25903.34} C_VEL
LIN {X 0,Y 178.043,Z 305.374,A -85,B 0,C 180,E1 -25904.719,E2 -25904.719} C_VEL
LIN {X 0,Y 181.939,Z 292.753,A -85,B 0,C 180,E1 -25905.818,E2 -25905.818} C_VEL
LIN {X 0,Y 184.832,Z 279.608,A -85,B 0,C 180,E1 -25906.596,E2 -25906.596} C_VEL
LIN {X 0,Y 186.705,Z 264.91,A -85,B 0,C 180,E1 -25907.107,E2 -25907.107} C_VEL
LIN {X 0,Y 186.807,Z 262.894,A -85,B 0,C 180,E1 -25907.231,E2 -25907.231} C_VEL
LIN {X 0,Y 183.449,Z 256.064,A -85,B 0,C 180,E1 -25910.491,E2 -25910.491} C_VEL
LIN {X 0,Y 180.83,Z 251.049,A -85,B 0,C 180,E1 -25913.58,E2 -25913.58} C_VEL
LIN {X 0,Y 178.907,Z 247.362,A -85,B 0,C 180,E1 -25916.327,E2 -25916.327} C_VEL
LIN {X 0,Y 177.309,Z 244.444,A -85,B 0,C 180,E1 -25919.119,E2 -25919.119} C_VEL
LIN {X 0,Y 175.663,Z 241.293,A -85,B 0,C 180,E1 -25923.434,E2 -25923.434} C_VEL
LIN {X 0,Y 175.409,Z 240.354,A -85,B 0,C 180,E1 -25924.597,E2 -25924.597} C_VEL
LIN {X 0,Y 174.786,Z 240.165,A -85,B 0,C 180,E1 -25931.599,E2 -25931.599} C_VEL
LIN {X 0,Y 175.208,Z 240.58,A -85,B 0,C 180,E1 -25934.179,E2 -25934.179} C_VEL
LIN {X 0,Y 176.862,Z 244.766,A -85,B 0,C 180,E1 -25939.613,E2 -25939.613} C_VEL
LIN {X 0,Y 177.676,Z 246.637,A -85,B 0,C 180,E1 -25941.282,E2 -25941.282} C_VEL
LIN {X 0,Y 179.606,Z 250.994,A -85,B 0,C 180,E1 -25944.497,E2 -25944.497} C_VEL
LIN {X 0,Y 181.69,Z 256.262,A -85,B 0,C 180,E1 -25947.378,E2 -25947.378} C_VEL
LIN {X 0,Y 184.076,Z 262.627,A -85,B 0,C 180,E1 -25950.153,E2 -25950.153} C_VEL
LIN {X 0,Y 186.302,Z 269.086,A -85,B 0,C 180,E1 -25952.43,E2 -25952.43} C_VEL
LIN {X 0,Y 184.411,Z 285.462,A -85,B 0,C 180,E1 -25953.025,E2 -25953.025} C_VEL
LIN {X 0,Y 181.667,Z 297.927,A -85,B 0,C 180,E1 -25953.6,E2 -25953.6} C_VEL
LIN {X 0,Y 177.918,Z 310.004,A -85,B 0,C 180,E1 -25954.452,E2 -25954.452} C_VEL
LIN {X 0,Y 172.993,Z 322.183,A -85,B 0,C 180,E1 -25955.657,E2 -25955.657} C_VEL
LIN {X 0,Y 167.458,Z 333.134,A -85,B 0,C 180,E1 -25957.116,E2 -25957.116} C_VEL
LIN {X 0,Y 162.063,Z 342.049,A -85,B 0,C 180,E1 -25958.685,E2 -25958.685} C_VEL
LIN {X 0,Y 155.67,Z 351.22,A -85,B 0,C 180,E1 -25960.868,E2 -25960.868} C_VEL
LIN {X 0,Y 148.307,Z 360.177,A -85,B 0,C 180,E1 -25963.724,E2 -25963.724} C_VEL
LIN {X 0,Y 141.407,Z 367.432,A -85,B 0,C 180,E1 -25966.891,E2 -25966.891} C_VEL
LIN {X 0,Y 133.978,Z 374.129,A -85,B 0,C 180,E1 -25970.988,E2 -25970.988} C_VEL
LIN {X 0,Y 127.584,Z 379.288,A -85,B 0,C 180,E1 -25975.72,E2 -25975.72} C_VEL
LIN {X 0,Y 123.714,Z 382.04,A -85,B 0,C 180,E1 -25979.25,E2 -25979.25} C_VEL
LIN {X 0,Y 118.405,Z 385.131,A -85,B 0,C 180,E1 -25985.449,E2 -25985.449} C_VEL
